KUKA KRL program: EPS_2_25694_LG02_A_20260223033039.src

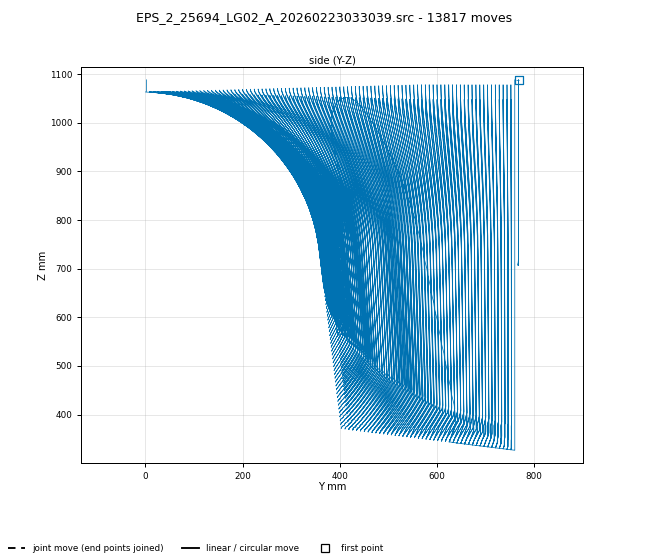
[picture p0: tool path of EPS_2_25694_LG02_A_20260223033039.src, 13817 of 13819 moves have a stored position in this frame; points joined in program order, loops and branches not executed]
&ACCESS RVP
&REL 4
&COMMENT QRS 19112012
&PARAM EDITMASK = *
DEF PART()
EXT BAS (BAS_COMMAND :IN,REAL :IN )
INT I
BAS (#INITMOV,0 )

;KUKA QRS Post kuka4.cps  Date:22-06-2017 !

File_ID=3045

QRS_PRE_INIT()

;Init var - Until changes are made in qrs_pre_init
Outlet_Square_prg=0
Inlet_1_Square_prg=0
Inlet_2_Square_prg=0
Inlet_3_Square_prg=0
Inlet_4_Square_prg=0
Inlet_5_Square_prg=0

Outlet_1={X 0.000, Y 562.000, Z 735.500, B 0.000, E1 0.000 }
Inlet_1={X 0.000, Y 562.000, Z 705.500, B 0.000, E1 182.000 }
Outlet_1_type=686
Inlet_1_type=686
;QRS#1=Sidecore dimensions
;QRS#2=675-27" Concrete
;QRS#3=675-27" Concrete
;QRS#4=
;QRS#5=
;QRS#6=
;QRS#7=
;QRS#8=
;QRS#9=S306-38L
;QRS#10=S306-38L
;QRS#11=
;QRS#12=
;QRS#13=
;QRS#14=
;QRS#15=
;QRS#16=1524x152x1524 5'
;QRS#17=EPS Height
;QRS#18=1078,5
;QRS#19=*
;QRS#20= UPDATED VERSION 22-06-2017
;QRS#21=*
Outlet_Square=0550
Inlet_1_Square=0550
Inlet_2_Square=0
Inlet_3_Square=0
Inlet_4_Square=0
Inlet_5_Square=0
Mill_Square=1
Outlet_Square_Prg=265
Inlet_1_Square_prg=265

QRS_INIT()

$ADVANCE=5

; T1
PTP {E1 173.043,E2 173.043}
PTP {X 0,Y 767.707,A -85,B 0,C 180,E1 173.043,E2 173.043,E3 0,E4 0,E5 0,E6 0}
QRS_SPEED_INIT()
LIN {X 0,Y 767.707,Z 1088.5,A -85,B 0,C 180,E1 173.043,E2 173.043,E3 0,E4 0,E5 0,E6 0} C_VEL
LIN {X 0,Y 767.707,Z 709.31,A -85,B 0,C 180,E1 173.043,E2 173.043} C_VEL
LIN {X 0,Y 767.734,Z 707.31,A -85,B 0,C 180,E1 173.192,E2 173.192} C_VEL
LIN {X 0,Y 767.794,Z 707.31,A -85,B 0,C 180,E1 173.458,E2 173.458} C_VEL
LIN {X 0,Y 767.812,Z 707.31,A -85,B 0,C 180,E1 177.201,E2 177.201} C_VEL
LIN {X 0,Y 767.838,Z 707.31,A -85,B 0,C 180,E1 180.933,E2 180.933} C_VEL
LIN {X 0,Y 767.834,Z 707.31,A -85,B 0,C 180,E1 184.668,E2 184.668} C_VEL
LIN {X 0,Y 767.857,Z 707.31,A -85,B 0,C 180,E1 188.423,E2 188.423} C_VEL
LIN {X 0,Y 767.828,Z 707.31,A -85,B 0,C 180,E1 192.215,E2 192.215} C_VEL
LIN {X 0,Y 767.83,Z 707.31,A -85,B 0,C 180,E1 196.204,E2 196.204} C_VEL
LIN {X 0,Y 767.77,Z 707.31,A -85,B 0,C 180,E1 199.988,E2 199.988} C_VEL
LIN {X 0,Y 767.749,Z 707.31,A -85,B 0,C 180,E1 204.013,E2 204.013} C_VEL
LIN {X 0,Y 767.749,Z 707.31,A -85,B 0,C 180,E1 208.167,E2 208.167} C_VEL
LIN {X 0,Y 767.324,Z 707.31,A -85,B 0,C 180,E1 210.324,E2 210.324} C_VEL
LIN {X 0,Y 767.754,Z 707.31,A -85,B 0,C 180,E1 212.49,E2 212.49} C_VEL
LIN {X 0,Y 767.43,Z 707.31,A -85,B 0,C 180,E1 213.85,E2 213.85} C_VEL
LIN {X 0,Y 767.706,Z 707.31,A -85,B 0,C 180,E1 217.094,E2 217.094} C_VEL
LIN {X 0,Y 767.087,Z 707.31,A -85,B 0,C 180,E1 220.03,E2 220.03} C_VEL
LIN {X 0,Y 767.533,Z 707.31,A -85,B 0,C 180,E1 221.88,E2 221.88} C_VEL
LIN {X 0,Y 767.581,Z 707.31,A -85,B 0,C 180,E1 222.891,E2 222.891} C_VEL
LIN {X 0,Y 767.581,Z 707.31,A -85,B 0,C 180,E1 227.109,E2 227.109} C_VEL
LIN {X 0,Y 767.53,Z 707.31,A -85,B 0,C 180,E1 228.12,E2 228.12} C_VEL
LIN {X 0,Y 767.102,Z 707.31,A -85,B 0,C 180,E1 230.553,E2 230.553} C_VEL
LIN {X 0,Y 767.692,Z 707.31,A -85,B 0,C 180,E1 232.964,E2 232.964} C_VEL
LIN {X 0,Y 767.598,Z 707.31,A -85,B 0,C 180,E1 236.132,E2 236.132} C_VEL
LIN {X 0,Y 767.614,Z 707.31,A -85,B 0,C 180,E1 237.503,E2 237.503} C_VEL
LIN {X 0,Y 767.641,Z 707.31,A -85,B 0,C 180,E1 239.69,E2 239.69} C_VEL
LIN {X 0,Y 767.411,Z 728.972,A -85,B 0,C 180,E1 240.873,E2 240.873} C_VEL
LIN {X 0,Y 767.537,Z 761.794,A -85,B 0,C 180,E1 241.233,E2 241.233} C_VEL
LIN {X 0,Y 767.433,Z 775.287,A -85,B 0,C 180,E1 241.407,E2 241.407} C_VEL
LIN {X 0,Y 767.548,Z 791.125,A -85,B 0,C 180,E1 241.677,E2 241.677} C_VEL
LIN {X 0,Y 767.449,Z 807.751,A -85,B 0,C 180,E1 242.019,E2 242.019} C_VEL
LIN {X 0,Y 767.663,Z 824.865,A -85,B 0,C 180,E1 242.456,E2 242.456} C_VEL
LIN {X 0,Y 767.66,Z 840.824,A -85,B 0,C 180,E1 242.921,E2 242.921} C_VEL
LIN {X 0,Y 767.553,Z 854.893,A -85,B 0,C 180,E1 243.38,E2 243.38} C_VEL
LIN {X 0,Y 767.694,Z 871.263,A -85,B 0,C 180,E1 243.998,E2 243.998} C_VEL
LIN {X 0,Y 767.655,Z 888.029,A -85,B 0,C 180,E1 244.706,E2 244.706} C_VEL
LIN {X 0,Y 767.705,Z 901.803,A -85,B 0,C 180,E1 245.351,E2 245.351} C_VEL
LIN {X 0,Y 767.712,Z 916.578,A -85,B 0,C 180,E1 246.114,E2 246.114} C_VEL
LIN {X 0,Y 767.693,Z 930.073,A -85,B 0,C 180,E1 246.876,E2 246.876} C_VEL
LIN {X 0,Y 767.691,Z 942.43,A -85,B 0,C 180,E1 247.634,E2 247.634} C_VEL
LIN {X 0,Y 767.701,Z 955.671,A -85,B 0,C 180,E1 248.523,E2 248.523} C_VEL
LIN {X 0,Y 767.718,Z 968.193,A -85,B 0,C 180,E1 249.439,E2 249.439} C_VEL
LIN {X 0,Y 767.619,Z 980.058,A -85,B 0,C 180,E1 250.38,E2 250.38} C_VEL
LIN {X 0,Y 767.656,Z 990.133,A -85,B 0,C 180,E1 251.245,E2 251.245} C_VEL
LIN {X 0,Y 767.778,Z 1000.684,A -85,B 0,C 180,E1 252.23,E2 252.23} C_VEL
LIN {X 0,Y 767.637,Z 1011.458,A -85,B 0,C 180,E1 253.326,E2 253.326} C_VEL
LIN {X 0,Y 767.699,Z 1020.421,A -85,B 0,C 180,E1 254.322,E2 254.322} C_VEL
LIN {X 0,Y 767.767,Z 1028.418,A -85,B 0,C 180,E1 255.29,E2 255.29} C_VEL
LIN {X 0,Y 767.624,Z 1037.824,A -85,B 0,C 180,E1 256.546,E2 256.546} C_VEL
LIN {X 0,Y 767.75,Z 1044.548,A -85,B 0,C 180,E1 257.545,E2 257.545} C_VEL
LIN {X 0,Y 767.749,Z 1048.907,A -85,B 0,C 180,E1 258.26,E2 258.26} C_VEL
LIN {X 0,Y 767.595,Z 1053.115,A -85,B 0,C 180,E1 258.971,E2 258.971} C_VEL
LIN {X 0,Y 767.579,Z 1059.347,A -85,B 0,C 180,E1 260.157,E2 260.157} C_VEL
LIN {X 0,Y 767.814,Z 1064.751,A -85,B 0,C 180,E1 261.341,E2 261.341} C_VEL
LIN {X 0,Y 767.552,Z 1069.482,A -85,B 0,C 180,E1 262.516,E2 262.516} C_VEL
LIN {X 0,Y 767.638,Z 1073.816,A -85,B 0,C 180,E1 263.832,E2 263.832} C_VEL
LIN {X 0,Y 767.832,Z 1075.822,A -85,B 0,C 180,E1 264.583,E2 264.583} C_VEL
LIN {X 0,Y 767.656,Z 1077.679,A -85,B 0,C 180,E1 265.331,E2 265.331} C_VEL
LIN {X 0,Y 767.554,Z 1079.934,A -85,B 0,C 180,E1 266.453,E2 266.453} C_VEL
LIN {X 0,Y 767.665,Z 1081.027,A -85,B 0,C 180,E1 267.201,E2 267.201} C_VEL
LIN {X 0,Y 767.713,Z 1082.196,A -85,B 0,C 180,E1 268.321,E2 268.321} C_VEL
LIN {X 0,Y 767.556,Z 1082.708,A -85,B 0,C 180,E1 269.067,E2 269.067} C_VEL
LIN {X 0,Y 767.7,Z 1082.68,A -85,B 0,C 180,E1 270.933,E2 270.933} C_VEL
LIN {X 0,Y 767.756,Z 1082.187,A -85,B 0,C 180,E1 271.679,E2 271.679} C_VEL
LIN {X 0,Y 767.525,Z 1081.053,A -85,B 0,C 180,E1 272.8,E2 272.8} C_VEL
LIN {X 0,Y 767.569,Z 1079.273,A -85,B 0,C 180,E1 273.921,E2 273.921} C_VEL
LIN {X 0,Y 767.76,Z 1077.66,A -85,B 0,C 180,E1 274.668,E2 274.668} C_VEL
LIN {X 0,Y 767.653,Z 1074.831,A -85,B 0,C 180,E1 275.793,E2 275.793} C_VEL
LIN {X 0,Y 767.602,Z 1072.628,A -85,B 0,C 180,E1 276.544,E2 276.544} C_VEL
LIN {X 0,Y 767.713,Z 1069.455,A -85,B 0,C 180,E1 277.483,E2 277.483} C_VEL
LIN {X 0,Y 767.824,Z 1067.577,A -85,B 0,C 180,E1 277.952,E2 277.952} C_VEL
LIN {X 0,Y 767.62,Z 1063.756,A -85,B 0,C 180,E1 278.897,E2 278.897} C_VEL
LIN {X 0,Y 767.559,Z 1058.195,A -85,B 0,C 180,E1 280.08,E2 280.08} C_VEL
LIN {X 0,Y 767.835,Z 1051.779,A -85,B 0,C 180,E1 281.263,E2 281.263} C_VEL
LIN {X 0,Y 767.624,Z 1044.562,A -85,B 0,C 180,E1 282.457,E2 282.457} C_VEL
LIN {X 0,Y 767.658,Z 1036.703,A -85,B 0,C 180,E1 283.612,E2 283.612} C_VEL
LIN {X 0,Y 767.821,Z 1029.879,A -85,B 0,C 180,E1 284.516,E2 284.516} C_VEL
LIN {X 0,Y 767.629,Z 1020.425,A -85,B 0,C 180,E1 285.679,E2 285.679} C_VEL
LIN {X 0,Y 767.731,Z 1009.175,A -85,B 0,C 180,E1 286.916,E2 286.916} C_VEL
LIN {X 0,Y 767.752,Z 999.435,A -85,B 0,C 180,E1 287.893,E2 287.893} C_VEL
LIN {X 0,Y 767.658,Z 988.765,A -85,B 0,C 180,E1 288.878,E2 288.878} C_VEL
LIN {X 0,Y 767.742,Z 977.061,A -85,B 0,C 180,E1 289.864,E2 289.864} C_VEL
LIN {X 0,Y 767.717,Z 964.937,A -85,B 0,C 180,E1 290.806,E2 290.806} C_VEL
LIN {X 0,Y 767.695,Z 954,A -85,B 0,C 180,E1 291.594,E2 291.594} C_VEL
LIN {X 0,Y 767.712,Z 940.407,A -85,B 0,C 180,E1 292.491,E2 292.491} C_VEL
LIN {X 0,Y 767.708,Z 926.801,A -85,B 0,C 180,E1 293.314,E2 293.314} C_VEL
LIN {X 0,Y 767.702,Z 913.125,A -85,B 0,C 180,E1 294.071,E2 294.071} C_VEL
LIN {X 0,Y 767.609,Z 898.313,A -85,B 0,C 180,E1 294.82,E2 294.82} C_VEL
LIN {X 0,Y 767.699,Z 884.655,A -85,B 0,C 180,E1 295.444,E2 295.444} C_VEL
LIN {X 0,Y 767.675,Z 869.452,A -85,B 0,C 180,E1 296.074,E2 296.074} C_VEL
LIN {X 0,Y 767.622,Z 855.716,A -85,B 0,C 180,E1 296.587,E2 296.587} C_VEL
LIN {X 0,Y 767.679,Z 837.478,A -85,B 0,C 180,E1 297.183,E2 297.183} C_VEL
LIN {X 0,Y 767.517,Z 820.546,A -85,B 0,C 180,E1 297.665,E2 297.665} C_VEL
LIN {X 0,Y 767.57,Z 810.446,A -85,B 0,C 180,E1 297.91,E2 297.91} C_VEL
LIN {X 0,Y 767.621,Z 801.596,A -85,B 0,C 180,E1 298.106,E2 298.106} C_VEL
LIN {X 0,Y 767.599,Z 787.938,A -85,B 0,C 180,E1 298.38,E2 298.38} C_VEL
LIN {X 0,Y 767.429,Z 775.319,A -85,B 0,C 180,E1 298.593,E2 298.593} C_VEL
LIN {X 0,Y 767.549,Z 757.089,A -85,B 0,C 180,E1 298.825,E2 298.825} C_VEL
LIN {X 0,Y 767.411,Z 729.388,A -85,B 0,C 180,E1 299.122,E2 299.122} C_VEL
LIN {X 0,Y 767.69,Z 707.31,A -85,B 0,C 180,E1 300.308,E2 300.308} C_VEL
LIN {X 0,Y 767.796,Z 707.31,A -85,B 0,C 180,E1 302.488,E2 302.488} C_VEL
LIN {X 0,Y 767.259,Z 707.31,A -85,B 0,C 180,E1 304.756,E2 304.756} C_VEL
LIN {X 0,Y 767.698,Z 707.31,A -85,B 0,C 180,E1 307.093,E2 307.093} C_VEL
LIN {X 0,Y 767.134,Z 707.31,A -85,B 0,C 180,E1 310.034,E2 310.034} C_VEL
LIN {X 0,Y 767.63,Z 707.31,A -85,B 0,C 180,E1 311.873,E2 311.873} C_VEL
LIN {X 0,Y 767.669,Z 707.31,A -85,B 0,C 180,E1 312.898,E2 312.898} C_VEL
LIN {X 0,Y 767.67,Z 707.31,A -85,B 0,C 180,E1 314.427,E2 314.427} C_VEL
LIN {X 0,Y 767.632,Z 707.31,A -85,B 0,C 180,E1 315.57,E2 315.57} C_VEL
LIN {X 0,Y 767.641,Z 707.31,A -85,B 0,C 180,E1 319.92,E2 319.92} C_VEL
LIN {X 0,Y 767.641,Z 707.31,A -85,B 0,C 180,E1 320.586,E2 320.586} C_VEL
LIN {X 0,Y 767.2,Z 707.31,A -85,B 0,C 180,E1 322.956,E2 322.956} C_VEL
LIN {X 0,Y 767.714,Z 707.31,A -85,B 0,C 180,E1 325.268,E2 325.268} C_VEL
LIN {X 0,Y 767.762,Z 707.31,A -85,B 0,C 180,E1 329.62,E2 329.62} C_VEL
LIN {X 0,Y 767.769,Z 707.31,A -85,B 0,C 180,E1 333.539,E2 333.539} C_VEL
LIN {X 0,Y 767.759,Z 707.31,A -85,B 0,C 180,E1 333.929,E2 333.929} C_VEL
LIN {X 0,Y 767.758,Z 707.31,A -85,B 0,C 180,E1 338.014,E2 338.014} C_VEL
LIN {X 0,Y 767.79,Z 707.31,A -85,B 0,C 180,E1 341.986,E2 341.986} C_VEL
LIN {X 0,Y 767.525,Z 707.31,A -85,B 0,C 180,E1 343.931,E2 343.931} C_VEL
LIN {X 0,Y 767.673,Z 707.31,A -85,B 0,C 180,E1 345.866,E2 345.866} C_VEL
LIN {X 0,Y 767.85,Z 707.31,A -85,B 0,C 180,E1 349.687,E2 349.687} C_VEL
LIN {X 0,Y 767.871,Z 707.31,A -85,B 0,C 180,E1 353.458,E2 353.458} C_VEL
LIN {X 0,Y 767.845,Z 707.31,A -85,B 0,C 180,E1 357.201,E2 357.201} C_VEL
LIN {X 0,Y 767.813,Z 707.31,A -85,B 0,C 180,E1 360.933,E2 360.933} C_VEL
LIN {X 0,Y 767.808,Z 707.31,A -85,B 0,C 180,E1 364.668,E2 364.668} C_VEL
LIN {X 0,Y 767.797,Z 707.31,A -85,B 0,C 180,E1 368.424,E2 368.424} C_VEL
LIN {X 0,Y 767.811,Z 707.31,A -85,B 0,C 180,E1 372.216,E2 372.216} C_VEL
LIN {X 0,Y 767.847,Z 707.31,A -85,B 0,C 180,E1 376.209,E2 376.209} C_VEL
LIN {X 0,Y 767.467,Z 707.31,A -85,B 0,C 180,E1 379.996,E2 379.996} C_VEL
LIN {X 0,Y 767.321,Z 707.31,A -85,B 0,C 180,E1 381.999,E2 381.999} C_VEL
LIN {X 0,Y 767.24,Z 707.31,A -85,B 0,C 180,E1 384.03,E2 384.03} C_VEL
LIN {X 0,Y 767.58,Z 707.31,A -85,B 0,C 180,E1 386.078,E2 386.078} C_VEL
LIN {X 0,Y 767.754,Z 707.31,A -85,B 0,C 180,E1 390.379,E2 390.379} C_VEL
LIN {X 0,Y 767.374,Z 707.31,A -85,B 0,C 180,E1 393.844,E2 393.844} C_VEL
LIN {X 0,Y 767.676,Z 707.31,A -85,B 0,C 180,E1 394.734,E2 394.734} C_VEL
LIN {X 0,Y 767.196,Z 707.31,A -85,B 0,C 180,E1 397.064,E2 397.064} C_VEL
LIN {X 0,Y 767.661,Z 707.31,A -85,B 0,C 180,E1 399.412,E2 399.412} C_VEL
LIN {X 0,Y 767.663,Z 707.31,A -85,B 0,C 180,E1 400.082,E2 400.082} C_VEL
LIN {X 0,Y 767.636,Z 707.31,A -85,B 0,C 180,E1 404.43,E2 404.43} C_VEL
LIN {X 0,Y 767.465,Z 707.31,A -85,B 0,C 180,E1 405.558,E2 405.558} C_VEL
LIN {X 0,Y 767.675,Z 707.31,A -85,B 0,C 180,E1 409.918,E2 409.918} C_VEL
LIN {X 0,Y 767.742,Z 707.31,A -85,B 0,C 180,E1 410.593,E2 410.593} C_VEL
LIN {X 0,Y 767.651,Z 707.31,A -85,B 0,C 180,E1 412.962,E2 412.962} C_VEL
LIN {X 0,Y 767.133,Z 707.31,A -85,B 0,C 180,E1 415.238,E2 415.238} C_VEL
LIN {X 0,Y 767.859,Z 707.31,A -85,B 0,C 180,E1 418.652,E2 418.652} C_VEL
LIN {X 0,Y 766.583,Z 707.31,A -85,B 0,C 180,E1 418.851,E2 418.851} C_VEL
LIN {X 0,Y 766.332,Z 707.453,A -85,B 0,C 180,E1 418.872,E2 418.872} C_VEL
LIN {X 0,Y 767.228,Z 716.962,A -85,B 0,C 180,E1 419.009,E2 419.009} C_VEL
LIN {X 0,Y 767.514,Z 728.846,A -85,B 0,C 180,E1 419.15,E2 419.15} C_VEL
LIN {X 0,Y 767.577,Z 744.469,A -85,B 0,C 180,E1 419.354,E2 419.354} C_VEL
LIN {X 0,Y 767.448,Z 760.576,A -85,B 0,C 180,E1 419.617,E2 419.617} C_VEL
LIN {X 0,Y 767.544,Z 778.604,A -85,B 0,C 180,E1 419.999,E2 419.999} C_VEL
LIN {X 0,Y 767.515,Z 791.795,A -85,B 0,C 180,E1 420.32,E2 420.32} C_VEL
LIN {X 0,Y 767.646,Z 810.803,A -85,B 0,C 180,E1 420.875,E2 420.875} C_VEL
LIN {X 0,Y 767.539,Z 825.708,A -85,B 0,C 180,E1 421.364,E2 421.364} C_VEL
LIN {X 0,Y 767.659,Z 841.503,A -85,B 0,C 180,E1 421.961,E2 421.961} C_VEL
LIN {X 0,Y 767.652,Z 857.144,A -85,B 0,C 180,E1 422.619,E2 422.619} C_VEL
LIN {X 0,Y 767.699,Z 872.8,A -85,B 0,C 180,E1 423.357,E2 423.357} C_VEL
LIN {X 0,Y 767.696,Z 886.598,A -85,B 0,C 180,E1 424.069,E2 424.069} C_VEL
LIN {X 0,Y 767.675,Z 900.841,A -85,B 0,C 180,E1 424.877,E2 424.877} C_VEL
LIN {X 0,Y 767.698,Z 912.552,A -85,B 0,C 180,E1 425.598,E2 425.598} C_VEL
LIN {X 0,Y 767.712,Z 925.914,A -85,B 0,C 180,E1 426.496,E2 426.496} C_VEL
LIN {X 0,Y 767.737,Z 938.055,A -85,B 0,C 180,E1 427.383,E2 427.383} C_VEL
LIN {X 0,Y 767.685,Z 949.6,A -85,B 0,C 180,E1 428.298,E2 428.298} C_VEL
LIN {X 0,Y 767.77,Z 960.082,A -85,B 0,C 180,E1 429.198,E2 429.198} C_VEL
LIN {X 0,Y 767.697,Z 971.428,A -85,B 0,C 180,E1 430.258,E2 430.258} C_VEL
LIN {X 0,Y 767.651,Z 981.132,A -85,B 0,C 180,E1 431.245,E2 431.245} C_VEL
LIN {X 0,Y 767.822,Z 991.022,A -85,B 0,C 180,E1 432.354,E2 432.354} C_VEL
LIN {X 0,Y 767.594,Z 999.985,A -85,B 0,C 180,E1 433.446,E2 433.446} C_VEL
LIN {X 0,Y 767.611,Z 1007.914,A -85,B 0,C 180,E1 434.514,E2 434.514} C_VEL
LIN {X 0,Y 767.808,Z 1015.644,A -85,B 0,C 180,E1 435.676,E2 435.676} C_VEL
LIN {X 0,Y 767.569,Z 1022.576,A -85,B 0,C 180,E1 436.824,E2 436.824} C_VEL
LIN {X 0,Y 767.623,Z 1028.911,A -85,B 0,C 180,E1 438.02,E2 438.02} C_VEL
LIN {X 0,Y 767.827,Z 1033.324,A -85,B 0,C 180,E1 438.975,E2 438.975} C_VEL
LIN {X 0,Y 767.639,Z 1036.336,A -85,B 0,C 180,E1 439.684,E2 439.684} C_VEL
LIN {X 0,Y 767.554,Z 1040.012,A -85,B 0,C 180,E1 440.63,E2 440.63} C_VEL
LIN {X 0,Y 767.677,Z 1043.168,A -85,B 0,C 180,E1 441.575,E2 441.575} C_VEL
LIN {X 0,Y 767.804,Z 1044.49,A -85,B 0,C 180,E1 442.048,E2 442.048} C_VEL
LIN {X 0,Y 767.778,Z 1045.777,A -85,B 0,C 180,E1 442.518,E2 442.518} C_VEL
LIN {X 0,Y 767.584,Z 1048.049,A -85,B 0,C 180,E1 443.456,E2 443.456} C_VEL
LIN {X 0,Y 767.578,Z 1049.627,A -85,B 0,C 180,E1 444.207,E2 444.207} C_VEL
LIN {X 0,Y 767.792,Z 1051.269,A -85,B 0,C 180,E1 445.332,E2 445.332} C_VEL
LIN {X 0,Y 767.688,Z 1052.025,A -85,B 0,C 180,E1 446.08,E2 446.08} C_VEL
LIN {X 0,Y 767.517,Z 1052.766,A -85,B 0,C 180,E1 447.2,E2 447.2} C_VEL
LIN {X 0,Y 767.839,Z 1052.603,A -85,B 0,C 180,E1 449.067,E2 449.067} C_VEL
LIN {X 0,Y 767.684,Z 1051.712,A -85,B 0,C 180,E1 450.187,E2 450.187} C_VEL
LIN {X 0,Y 767.839,Z 1049.617,A -85,B 0,C 180,E1 451.679,E2 451.679} C_VEL
LIN {X 0,Y 767.587,Z 1047.326,A -85,B 0,C 180,E1 452.8,E2 452.8} C_VEL
LIN {X 0,Y 767.682,Z 1043.303,A -85,B 0,C 180,E1 454.295,E2 454.295} C_VEL
LIN {X 0,Y 767.813,Z 1040.757,A -85,B 0,C 180,E1 455.042,E2 455.042} C_VEL
LIN {X 0,Y 767.73,Z 1039.519,A -85,B 0,C 180,E1 455.417,E2 455.417} C_VEL
LIN {X 0,Y 767.568,Z 1034.048,A -85,B 0,C 180,E1 456.792,E2 456.792} C_VEL
LIN {X 0,Y 767.782,Z 1028.581,A -85,B 0,C 180,E1 457.953,E2 457.953} C_VEL
LIN {X 0,Y 767.744,Z 1024.81,A -85,B 0,C 180,E1 458.66,E2 458.66} C_VEL
LIN {X 0,Y 767.59,Z 1020.908,A -85,B 0,C 180,E1 459.37,E2 459.37} C_VEL
LIN {X 0,Y 767.566,Z 1015.193,A -85,B 0,C 180,E1 460.317,E2 460.317} C_VEL
LIN {X 0,Y 767.802,Z 1007.156,A -85,B 0,C 180,E1 461.501,E2 461.501} C_VEL
LIN {X 0,Y 767.587,Z 998.194,A -85,B 0,C 180,E1 462.697,E2 462.697} C_VEL
LIN {X 0,Y 767.586,Z 989.678,A -85,B 0,C 180,E1 463.725,E2 463.725} C_VEL
LIN {X 0,Y 767.795,Z 978.848,A -85,B 0,C 180,E1 464.902,E2 464.902} C_VEL
LIN {X 0,Y 767.649,Z 968.142,A -85,B 0,C 180,E1 465.97,E2 465.97} C_VEL
LIN {X 0,Y 767.685,Z 957.768,A -85,B 0,C 180,E1 466.917,E2 466.917} C_VEL
LIN {X 0,Y 767.774,Z 947.684,A -85,B 0,C 180,E1 467.77,E2 467.77} C_VEL
LIN {X 0,Y 767.697,Z 935.041,A -85,B 0,C 180,E1 468.754,E2 468.754} C_VEL
LIN {X 0,Y 767.717,Z 922.969,A -85,B 0,C 180,E1 469.617,E2 469.617} C_VEL
LIN {X 0,Y 767.739,Z 910.052,A -85,B 0,C 180,E1 470.467,E2 470.467} C_VEL
LIN {X 0,Y 767.713,Z 896.37,A -85,B 0,C 180,E1 471.293,E2 471.293} C_VEL
LIN {X 0,Y 767.691,Z 882.652,A -85,B 0,C 180,E1 472.051,E2 472.051} C_VEL
LIN {X 0,Y 767.715,Z 868.914,A -85,B 0,C 180,E1 472.744,E2 472.744} C_VEL
LIN {X 0,Y 767.701,Z 853.646,A -85,B 0,C 180,E1 473.441,E2 473.441} C_VEL
LIN {X 0,Y 767.559,Z 838.183,A -85,B 0,C 180,E1 474.081,E2 474.081} C_VEL
LIN {X 0,Y 767.686,Z 823.019,A -85,B 0,C 180,E1 474.632,E2 474.632} C_VEL
LIN {X 0,Y 767.65,Z 807.174,A -85,B 0,C 180,E1 475.148,E2 475.148} C_VEL
LIN {X 0,Y 767.562,Z 793.513,A -85,B 0,C 180,E1 475.542,E2 475.542} C_VEL
LIN {X 0,Y 767.685,Z 773.931,A -85,B 0,C 180,E1 476.011,E2 476.011} C_VEL
LIN {X 0,Y 767.51,Z 756.999,A -85,B 0,C 180,E1 476.354,E2 476.354} C_VEL
LIN {X 0,Y 767.504,Z 749.285,A -85,B 0,C 180,E1 476.48,E2 476.48} C_VEL
LIN {X 0,Y 767.595,Z 739.533,A -85,B 0,C 180,E1 476.623,E2 476.623} C_VEL
LIN {X 0,Y 767.474,Z 719.835,A -85,B 0,C 180,E1 476.861,E2 476.861} C_VEL
LIN {X 0,Y 767.332,Z 713.145,A -85,B 0,C 180,E1 476.936,E2 476.936} C_VEL
LIN {X 0,Y 766.479,Z 708.854,A -85,B 0,C 180,E1 477.017,E2 477.017} C_VEL
LIN {X 0,Y 766.257,Z 707.31,A -85,B 0,C 180,E1 477.063,E2 477.063} C_VEL
LIN {X 0,Y 766.793,Z 707.31,A -85,B 0,C 180,E1 477.102,E2 477.102} C_VEL
LIN {X 0,Y 767.511,Z 707.31,A -85,B 0,C 180,E1 477.191,E2 477.191} C_VEL
LIN {X 0,Y 767.758,Z 707.31,A -85,B 0,C 180,E1 477.693,E2 477.693} C_VEL
LIN {X 0,Y 767.795,Z 707.31,A -85,B 0,C 180,E1 480.384,E2 480.384} C_VEL
LIN {X 0,Y 767.697,Z 707.31,A -85,B 0,C 180,E1 484.733,E2 484.733} C_VEL
LIN {X 0,Y 767.22,Z 707.31,A -85,B 0,C 180,E1 487.062,E2 487.062} C_VEL
LIN {X 0,Y 767.7,Z 707.31,A -85,B 0,C 180,E1 489.41,E2 489.41} C_VEL
LIN {X 0,Y 767.687,Z 707.31,A -85,B 0,C 180,E1 490.084,E2 490.084} C_VEL
LIN {X 0,Y 767.469,Z 707.31,A -85,B 0,C 180,E1 494.442,E2 494.442} C_VEL
LIN {X 0,Y 767.64,Z 707.31,A -85,B 0,C 180,E1 495.57,E2 495.57} C_VEL
LIN {X 0,Y 767.663,Z 707.31,A -85,B 0,C 180,E1 499.919,E2 499.919} C_VEL
LIN {X 0,Y 767.648,Z 707.31,A -85,B 0,C 180,E1 500.587,E2 500.587} C_VEL
LIN {X 0,Y 767.199,Z 707.31,A -85,B 0,C 180,E1 502.956,E2 502.956} C_VEL
LIN {X 0,Y 767.684,Z 707.31,A -85,B 0,C 180,E1 505.266,E2 505.266} C_VEL
LIN {X 0,Y 767.764,Z 707.31,A -85,B 0,C 180,E1 509.62,E2 509.62} C_VEL
LIN {X 0,Y 767.79,Z 707.31,A -85,B 0,C 180,E1 513.536,E2 513.536} C_VEL
LIN {X 0,Y 767.787,Z 707.31,A -85,B 0,C 180,E1 513.93,E2 513.93} C_VEL
LIN {X 0,Y 767.808,Z 707.31,A -85,B 0,C 180,E1 518.016,E2 518.016} C_VEL
LIN {X 0,Y 767.827,Z 707.31,A -85,B 0,C 180,E1 521.986,E2 521.986} C_VEL
LIN {X 0,Y 767.5,Z 707.31,A -85,B 0,C 180,E1 523.93,E2 523.93} C_VEL
LIN {X 0,Y 767.615,Z 707.31,A -85,B 0,C 180,E1 525.865,E2 525.865} C_VEL
LIN {X 0,Y 767.793,Z 707.31,A -85,B 0,C 180,E1 529.686,E2 529.686} C_VEL
LIN {X 0,Y 767.734,Z 707.31,A -85,B 0,C 180,E1 533.192,E2 533.192} C_VEL
LIN {X 0,Y 767.795,Z 709.31,A -85,B 0,C 180,E1 533.341,E2 533.341} C_VEL
LIN {X 0,Y 767.795,Z 1088.5,A -85,B 0,C 180,E1 533.341,E2 533.341} C_VEL
LIN {X 0,Y 767.795,Z 1088.5,A -85,B 0,C 180,E1 533.341,E2 533.341}

QRS_NEXT_CUT()
PTP {E1 537.319,E2 537.319}
PTP {X 0,Y 759.843,A -85,B 0,C 180,E1 537.319,E2 537.319,E3 0,E4 0,E5 0,E6 0}
QRS_SPEED_INIT()
LIN {X 0,Y 759.843,Z 1088.5,A -85,B 0,C 180,E1 537.319,E2 537.319,E3 0,E4 0,E5 0,E6 0} C_VEL
LIN {X 0,Y 759.843,Z 336.65,A -85,B 0,C 180,E1 537.319,E2 537.319} C_VEL
LIN {X 0,Y 759.843,Z 328.572,A -85,B 0,C 180,E1 537.319,E2 537.319} C_VEL
LIN {X 0,Y 759.843,Z 326.572,A -85,B 0,C 180,E1 537.169,E2 537.169} C_VEL
LIN {X 0,Y 759.893,Z 326.569,A -85,B 0,C 180,E1 534.564,E2 534.564} C_VEL
LIN {X 0,Y 759.866,Z 326.575,A -85,B 0,C 180,E1 531.601,E2 531.601} C_VEL
LIN {X 0,Y 759.843,Z 326.572,A -85,B 0,C 180,E1 529.077,E2 529.077} C_VEL
LIN {X 0,Y 759.889,Z 326.569,A -85,B 0,C 180,E1 526.454,E2 526.454} C_VEL
LIN {X 0,Y 759.869,Z 326.575,A -85,B 0,C 180,E1 523.487,E2 523.487} C_VEL
LIN {X 0,Y 759.844,Z 326.572,A -85,B 0,C 180,E1 520.953,E2 520.953} C_VEL
LIN {X 0,Y 759.881,Z 326.569,A -85,B 0,C 180,E1 518.381,E2 518.381} C_VEL
LIN {X 0,Y 759.869,Z 326.575,A -85,B 0,C 180,E1 515.346,E2 515.346} C_VEL
LIN {X 0,Y 759.844,Z 326.572,A -85,B 0,C 180,E1 512.818,E2 512.818} C_VEL
LIN {X 0,Y 759.879,Z 326.569,A -85,B 0,C 180,E1 510.259,E2 510.259} C_VEL
LIN {X 0,Y 759.872,Z 326.575,A -85,B 0,C 180,E1 507.229,E2 507.229} C_VEL
LIN {X 0,Y 759.845,Z 326.572,A -85,B 0,C 180,E1 504.673,E2 504.673} C_VEL
LIN {X 0,Y 759.898,Z 326.568,A -85,B 0,C 180,E1 501.989,E2 501.989} C_VEL
LIN {X 0,Y 759.869,Z 326.575,A -85,B 0,C 180,E1 499.052,E2 499.052} C_VEL
LIN {X 0,Y 759.846,Z 326.571,A -85,B 0,C 180,E1 496.51,E2 496.51} C_VEL
LIN {X 0,Y 759.898,Z 326.568,A -85,B 0,C 180,E1 493.857,E2 493.857} C_VEL
LIN {X 0,Y 759.873,Z 326.576,A -85,B 0,C 180,E1 490.942,E2 490.942} C_VEL
LIN {X 0,Y 759.846,Z 326.573,A -85,B 0,C 180,E1 488.397,E2 488.397} C_VEL
LIN {X 0,Y 759.894,Z 326.569,A -85,B 0,C 180,E1 485.748,E2 485.748} C_VEL
LIN {X 0,Y 759.868,Z 326.579,A -85,B 0,C 180,E1 482.77,E2 482.77} C_VEL
LIN {X 0,Y 759.846,Z 326.656,A -85,B 0,C 180,E1 482.25,E2 482.25} C_VEL
LIN {X 0,Y 759.884,Z 347.643,A -85,B 0,C 180,E1 480.755,E2 480.755} C_VEL
LIN {X 0,Y 759.912,Z 584.911,A -85,B 0,C 180,E1 478.177,E2 478.177} C_VEL
LIN {X 0,Y 759.916,Z 736.017,A -85,B 0,C 180,E1 476.55,E2 476.55} C_VEL
LIN {X 0,Y 759.9,Z 759.461,A -85,B 0,C 180,E1 476.182,E2 476.182} C_VEL
LIN {X 0,Y 759.903,Z 781.523,A -85,B 0,C 180,E1 475.701,E2 475.701} C_VEL
LIN {X 0,Y 759.898,Z 801.218,A -85,B 0,C 180,E1 475.172,E2 475.172} C_VEL
LIN {X 0,Y 759.919,Z 824.386,A -85,B 0,C 180,E1 474.421,E2 474.421} C_VEL
LIN {X 0,Y 759.916,Z 844.946,A -85,B 0,C 180,E1 473.619,E2 473.619} C_VEL
LIN {X 0,Y 759.913,Z 864.955,A -85,B 0,C 180,E1 472.724,E2 472.724} C_VEL
LIN {X 0,Y 759.91,Z 887,A -85,B 0,C 180,E1 471.578,E2 471.578} C_VEL
LIN {X 0,Y 759.916,Z 905.657,A -85,B 0,C 180,E1 470.471,E2 470.471} C_VEL
LIN {X 0,Y 759.908,Z 925.564,A -85,B 0,C 180,E1 469.125,E2 469.125} C_VEL
LIN {X 0,Y 759.913,Z 942.712,A -85,B 0,C 180,E1 467.814,E2 467.814} C_VEL
LIN {X 0,Y 759.912,Z 959.488,A -85,B 0,C 180,E1 466.355,E2 466.355} C_VEL
LIN {X 0,Y 759.897,Z 973.888,A -85,B 0,C 180,E1 464.946,E2 464.946} C_VEL
LIN {X 0,Y 759.908,Z 988.501,A -85,B 0,C 180,E1 463.313,E2 463.313} C_VEL
LIN {X 0,Y 759.906,Z 1000.009,A -85,B 0,C 180,E1 461.845,E2 461.845} C_VEL
LIN {X 0,Y 759.912,Z 1012.038,A -85,B 0,C 180,E1 460.079,E2 460.079} C_VEL
LIN {X 0,Y 759.9,Z 1021.248,A -85,B 0,C 180,E1 458.475,E2 458.475} C_VEL
LIN {X 0,Y 759.894,Z 1029.42,A -85,B 0,C 180,E1 456.801,E2 456.801} C_VEL
LIN {X 0,Y 759.914,Z 1036.478,A -85,B 0,C 180,E1 454.982,E2 454.982} C_VEL
LIN {X 0,Y 759.893,Z 1041.296,A -85,B 0,C 180,E1 453.395,E2 453.395} C_VEL
LIN {X 0,Y 759.914,Z 1045.436,A -85,B 0,C 180,E1 451.508,E2 451.508} C_VEL
LIN {X 0,Y 759.902,Z 1047.622,A -85,B 0,C 180,E1 449.774,E2 449.774} C_VEL
LIN {X 0,Y 759.911,Z 1048.5,A -85,B 0,C 180,E1 447.964,E2 447.964} C_VEL
LIN {X 0,Y 759.903,Z 1047.636,A -85,B 0,C 180,E1 446.152,E2 446.152} C_VEL
LIN {X 0,Y 759.912,Z 1045.563,A -85,B 0,C 180,E1 444.488,E2 444.488} C_VEL
LIN {X 0,Y 759.895,Z 1041.501,A -85,B 0,C 180,E1 442.591,E2 442.591} C_VEL
LIN {X 0,Y 759.914,Z 1036.69,A -85,B 0,C 180,E1 440.992,E2 440.992} C_VEL
LIN {X 0,Y 759.893,Z 1029.632,A -85,B 0,C 180,E1 439.154,E2 439.154} C_VEL
LIN {X 0,Y 759.904,Z 1021.383,A -85,B 0,C 180,E1 437.461,E2 437.461} C_VEL
LIN {X 0,Y 759.912,Z 1012.276,A -85,B 0,C 180,E1 435.871,E2 435.871} C_VEL
LIN {X 0,Y 759.907,Z 1000.391,A -85,B 0,C 180,E1 434.116,E2 434.116} C_VEL
LIN {X 0,Y 759.908,Z 988.697,A -85,B 0,C 180,E1 432.621,E2 432.621} C_VEL
LIN {X 0,Y 759.903,Z 973.001,A -85,B 0,C 180,E1 430.875,E2 430.875} C_VEL
LIN {X 0,Y 759.909,Z 959.029,A -85,B 0,C 180,E1 429.512,E2 429.512} C_VEL
LIN {X 0,Y 759.915,Z 940.673,A -85,B 0,C 180,E1 427.935,E2 427.935} C_VEL
LIN {X 0,Y 759.917,Z 923.41,A -85,B 0,C 180,E1 426.627,E2 426.627} C_VEL
LIN {X 0,Y 759.914,Z 903.513,A -85,B 0,C 180,E1 425.306,E2 425.306} C_VEL
LIN {X 0,Y 759.91,Z 885.071,A -85,B 0,C 180,E1 424.223,E2 424.223} C_VEL
LIN {X 0,Y 759.915,Z 862.835,A -85,B 0,C 180,E1 423.087,E2 423.087} C_VEL
LIN {X 0,Y 759.918,Z 843.709,A -85,B 0,C 180,E1 422.239,E2 422.239} C_VEL
LIN {X 0,Y 759.913,Z 820.69,A -85,B 0,C 180,E1 421.359,E2 421.359} C_VEL
LIN {X 0,Y 759.903,Z 799.673,A -85,B 0,C 180,E1 420.693,E2 420.693} C_VEL
LIN {X 0,Y 759.9,Z 779.134,A -85,B 0,C 180,E1 420.15,E2 420.15} C_VEL
LIN {X 0,Y 759.908,Z 753.73,A -85,B 0,C 180,E1 419.629,E2 419.629} C_VEL
LIN {X 0,Y 759.917,Z 733.55,A -85,B 0,C 180,E1 419.329,E2 419.329} C_VEL
LIN {X 0,Y 759.917,Z 462.351,A -85,B 0,C 180,E1 416.411,E2 416.411} C_VEL
LIN {X 0,Y 759.883,Z 347.478,A -85,B 0,C 180,E1 415.152,E2 415.152} C_VEL
LIN {X 0,Y 759.844,Z 326.576,A -85,B 0,C 180,E1 413.644,E2 413.644} C_VEL
LIN {X 0,Y 759.867,Z 326.576,A -85,B 0,C 180,E1 411.121,E2 411.121} C_VEL
LIN {X 0,Y 759.892,Z 326.569,A -85,B 0,C 180,E1 408.139,E2 408.139} C_VEL
LIN {X 0,Y 759.844,Z 326.572,A -85,B 0,C 180,E1 405.498,E2 405.498} C_VEL
LIN {X 0,Y 759.868,Z 326.575,A -85,B 0,C 180,E1 402.971,E2 402.971} C_VEL
LIN {X 0,Y 759.884,Z 326.569,A -85,B 0,C 180,E1 399.951,E2 399.951} C_VEL
LIN {X 0,Y 759.843,Z 326.573,A -85,B 0,C 180,E1 397.347,E2 397.347} C_VEL
LIN {X 0,Y 759.87,Z 326.574,A -85,B 0,C 180,E1 394.805,E2 394.805} C_VEL
LIN {X 0,Y 759.877,Z 326.569,A -85,B 0,C 180,E1 391.759,E2 391.759} C_VEL
LIN {X 0,Y 759.843,Z 326.572,A -85,B 0,C 180,E1 389.223,E2 389.223} C_VEL
LIN {X 0,Y 759.868,Z 326.575,A -85,B 0,C 180,E1 386.686,E2 386.686} C_VEL
LIN {X 0,Y 759.882,Z 326.569,A -85,B 0,C 180,E1 383.662,E2 383.662} C_VEL
LIN {X 0,Y 759.842,Z 326.572,A -85,B 0,C 180,E1 381.054,E2 381.054} C_VEL
LIN {X 0,Y 759.865,Z 326.575,A -85,B 0,C 180,E1 378.569,E2 378.569} C_VEL
LIN {X 0,Y 759.888,Z 326.569,A -85,B 0,C 180,E1 375.571,E2 375.571} C_VEL
LIN {X 0,Y 759.843,Z 326.572,A -85,B 0,C 180,E1 373.004,E2 373.004} C_VEL
LIN {X 0,Y 759.855,Z 326.575,A -85,B 0,C 180,E1 370.539,E2 370.539} C_VEL
LIN {X 0,Y 759.916,Z 326.569,A -85,B 0,C 180,E1 367.637,E2 367.637} C_VEL
LIN {X 0,Y 759.844,Z 326.572,A -85,B 0,C 180,E1 364.907,E2 364.907} C_VEL
LIN {X 0,Y 759.854,Z 326.575,A -85,B 0,C 180,E1 362.413,E2 362.413} C_VEL
LIN {X 0,Y 759.918,Z 326.57,A -85,B 0,C 180,E1 359.548,E2 359.548} C_VEL
LIN {X 0,Y 759.846,Z 326.571,A -85,B 0,C 180,E1 356.832,E2 356.832} C_VEL
LIN {X 0,Y 759.849,Z 326.574,A -85,B 0,C 180,E1 354.336,E2 354.336} C_VEL
LIN {X 0,Y 759.916,Z 326.572,A -85,B 0,C 180,E1 351.525,E2 351.525} C_VEL
LIN {X 0,Y 759.849,Z 326.571,A -85,B 0,C 180,E1 348.77,E2 348.77} C_VEL
LIN {X 0,Y 759.844,Z 326.574,A -85,B 0,C 180,E1 346.298,E2 346.298} C_VEL
LIN {X 0,Y 759.915,Z 326.577,A -85,B 0,C 180,E1 343.567,E2 343.567} C_VEL
LIN {X 0,Y 759.853,Z 326.571,A -85,B 0,C 180,E1 340.713,E2 340.713} C_VEL
LIN {X 0,Y 759.84,Z 326.573,A -85,B 0,C 180,E1 338.286,E2 338.286} C_VEL
LIN {X 0,Y 759.872,Z 326.575,A -85,B 0,C 180,E1 335.76,E2 335.76} C_VEL
LIN {X 0,Y 759.872,Z 326.57,A -85,B 0,C 180,E1 332.747,E2 332.747} C_VEL
LIN {X 0,Y 759.84,Z 326.573,A -85,B 0,C 180,E1 330.257,E2 330.257} C_VEL
LIN {X 0,Y 759.854,Z 326.575,A -85,B 0,C 180,E1 327.792,E2 327.792} C_VEL
LIN {X 0,Y 759.91,Z 326.57,A -85,B 0,C 180,E1 324.9,E2 324.9} C_VEL
LIN {X 0,Y 759.845,Z 326.572,A -85,B 0,C 180,E1 322.266,E2 322.266} C_VEL
LIN {X 0,Y 759.842,Z 326.574,A -85,B 0,C 180,E1 319.849,E2 319.849} C_VEL
LIN {X 0,Y 759.909,Z 326.578,A -85,B 0,C 180,E1 317.13,E2 317.13} C_VEL
LIN {X 0,Y 759.855,Z 326.571,A -85,B 0,C 180,E1 314.287,E2 314.287} C_VEL
LIN {X 0,Y 759.839,Z 326.574,A -85,B 0,C 180,E1 311.849,E2 311.849} C_VEL
LIN {X 0,Y 759.877,Z 326.577,A -85,B 0,C 180,E1 309.266,E2 309.266} C_VEL
LIN {X 0,Y 759.863,Z 326.573,A -85,B 0,C 180,E1 306.231,E2 306.231} C_VEL
LIN {X 0,Y 759.857,Z 326.883,A -85,B 0,C 180,E1 306.17,E2 306.17} C_VEL
LIN {X 0,Y 759.903,Z 363.722,A -85,B 0,C 180,E1 303.684,E2 303.684} C_VEL
LIN {X 0,Y 759.914,Z 377.344,A -85,B 0,C 180,E1 302.802,E2 302.802} C_VEL
LIN {X 0,Y 759.918,Z 632.42,A -85,B 0,C 180,E1 300.034,E2 300.034} C_VEL
LIN {X 0,Y 759.915,Z 765.994,A -85,B 0,C 180,E1 298.595,E2 298.595} C_VEL
LIN {X 0,Y 759.897,Z 790.301,A -85,B 0,C 180,E1 298.21,E2 298.21} C_VEL
LIN {X 0,Y 759.902,Z 811.683,A -85,B 0,C 180,E1 297.742,E2 297.742} C_VEL
LIN {X 0,Y 759.901,Z 831.086,A -85,B 0,C 180,E1 297.221,E2 297.221} C_VEL
LIN {X 0,Y 759.919,Z 853.739,A -85,B 0,C 180,E1 296.491,E2 296.491} C_VEL
LIN {X 0,Y 759.916,Z 875.252,A -85,B 0,C 180,E1 295.651,E2 295.651} C_VEL
LIN {X 0,Y 759.913,Z 894.66,A -85,B 0,C 180,E1 294.783,E2 294.783} C_VEL
LIN {X 0,Y 759.911,Z 917.061,A -85,B 0,C 180,E1 293.62,E2 293.62} C_VEL
LIN {X 0,Y 759.907,Z 935.706,A -85,B 0,C 180,E1 292.513,E2 292.513} C_VEL
LIN {X 0,Y 759.909,Z 955.524,A -85,B 0,C 180,E1 291.173,E2 291.173} C_VEL
LIN {X 0,Y 759.917,Z 972.885,A -85,B 0,C 180,E1 289.845,E2 289.845} C_VEL
LIN {X 0,Y 759.909,Z 989.391,A -85,B 0,C 180,E1 288.409,E2 288.409} C_VEL
LIN {X 0,Y 759.903,Z 1003.947,A -85,B 0,C 180,E1 286.984,E2 286.984} C_VEL
LIN {X 0,Y 759.915,Z 1018.836,A -85,B 0,C 180,E1 285.317,E2 285.317} C_VEL
LIN {X 0,Y 759.898,Z 1030.589,A -85,B 0,C 180,E1 283.812,E2 283.812} C_VEL
LIN {X 0,Y 759.901,Z 1042.785,A -85,B 0,C 180,E1 281.999,E2 281.999} C_VEL
LIN {X 0,Y 759.91,Z 1051.555,A -85,B 0,C 180,E1 280.462,E2 280.462} C_VEL
LIN {X 0,Y 759.89,Z 1060.073,A -85,B 0,C 180,E1 278.703,E2 278.703} C_VEL
LIN {X 0,Y 759.919,Z 1066.726,A -85,B 0,C 180,E1 276.953,E2 276.953} C_VEL
LIN {X 0,Y 759.906,Z 1071.51,A -85,B 0,C 180,E1 275.361,E2 275.361} C_VEL
LIN {X 0,Y 759.917,Z 1075.671,A -85,B 0,C 180,E1 273.395,E2 273.395} C_VEL
LIN {X 0,Y 759.899,Z 1077.63,A -85,B 0,C 180,E1 271.81,E2 271.81} C_VEL
LIN {X 0,Y 759.92,Z 1078.5,A -85,B 0,C 180,E1 270,E2 270} C_VEL
LIN {X 0,Y 759.899,Z 1077.63,A -85,B 0,C 180,E1 268.19,E2 268.19} C_VEL
LIN {X 0,Y 759.918,Z 1075.559,A -85,B 0,C 180,E1 266.53,E2 266.53} C_VEL
LIN {X 0,Y 759.906,Z 1071.51,A -85,B 0,C 180,E1 264.639,E2 264.639} C_VEL
LIN {X 0,Y 759.919,Z 1066.726,A -85,B 0,C 180,E1 263.047,E2 263.047} C_VEL
LIN {X 0,Y 759.892,Z 1059.729,A -85,B 0,C 180,E1 261.22,E2 261.22} C_VEL
LIN {X 0,Y 759.91,Z 1051.555,A -85,B 0,C 180,E1 259.538,E2 259.538} C_VEL
LIN {X 0,Y 759.901,Z 1042.786,A -85,B 0,C 180,E1 258.001,E2 258.001} C_VEL
LIN {X 0,Y 759.898,Z 1030.589,A -85,B 0,C 180,E1 256.188,E2 256.188} C_VEL
LIN {X 0,Y 759.917,Z 1018.833,A -85,B 0,C 180,E1 254.683,E2 254.683} C_VEL
LIN {X 0,Y 759.903,Z 1003.948,A -85,B 0,C 180,E1 253.016,E2 253.016} C_VEL
LIN {X 0,Y 759.909,Z 989.391,A -85,B 0,C 180,E1 251.591,E2 251.591} C_VEL
LIN {X 0,Y 759.911,Z 971.366,A -85,B 0,C 180,E1 250.035,E2 250.035} C_VEL
LIN {X 0,Y 759.913,Z 954.42,A -85,B 0,C 180,E1 248.746,E2 248.746} C_VEL
LIN {X 0,Y 759.909,Z 934.383,A -85,B 0,C 180,E1 247.405,E2 247.405} C_VEL
LIN {X 0,Y 759.91,Z 915.991,A -85,B 0,C 180,E1 246.32,E2 246.32} C_VEL
LIN {X 0,Y 759.912,Z 893.9,A -85,B 0,C 180,E1 245.182,E2 245.182} C_VEL
LIN {X 0,Y 759.916,Z 874.865,A -85,B 0,C 180,E1 244.332,E2 244.332} C_VEL
LIN {X 0,Y 759.916,Z 852.82,A -85,B 0,C 180,E1 243.475,E2 243.475} C_VEL
LIN {X 0,Y 759.901,Z 831.087,A -85,B 0,C 180,E1 242.779,E2 242.779} C_VEL
LIN {X 0,Y 759.902,Z 811.685,A -85,B 0,C 180,E1 242.258,E2 242.258} C_VEL
LIN {X 0,Y 759.899,Z 789.26,A -85,B 0,C 180,E1 241.768,E2 241.768} C_VEL
LIN {X 0,Y 759.917,Z 765.997,A -85,B 0,C 180,E1 241.405,E2 241.405} C_VEL
LIN {X 0,Y 759.899,Z 499.217,A -85,B 0,C 180,E1 238.53,E2 238.53} C_VEL
LIN {X 0,Y 759.911,Z 376.685,A -85,B 0,C 180,E1 237.173,E2 237.173} C_VEL
LIN {X 0,Y 759.853,Z 337.913,A -85,B 0,C 180,E1 234.582,E2 234.582} C_VEL
LIN {X 0,Y 759.861,Z 326.575,A -85,B 0,C 180,E1 233.784,E2 233.784} C_VEL
LIN {X 0,Y 759.887,Z 326.577,A -85,B 0,C 180,E1 230.808,E2 230.808} C_VEL
LIN {X 0,Y 759.841,Z 326.574,A -85,B 0,C 180,E1 228.252,E2 228.252} C_VEL
LIN {X 0,Y 759.85,Z 326.572,A -85,B 0,C 180,E1 225.779,E2 225.779} C_VEL
LIN {X 0,Y 759.913,Z 326.575,A -85,B 0,C 180,E1 222.968,E2 222.968} C_VEL
LIN {X 0,Y 759.847,Z 326.574,A -85,B 0,C 180,E1 220.249,E2 220.249} C_VEL
LIN {X 0,Y 759.841,Z 326.572,A -85,B 0,C 180,E1 217.823,E2 217.823} C_VEL
LIN {X 0,Y 759.9,Z 326.569,A -85,B 0,C 180,E1 215.193,E2 215.193} C_VEL
LIN {X 0,Y 759.862,Z 326.575,A -85,B 0,C 180,E1 212.293,E2 212.293} C_VEL
LIN {X 0,Y 759.84,Z 326.573,A -85,B 0,C 180,E1 209.83,E2 209.83} C_VEL
LIN {X 0,Y 759.863,Z 326.57,A -85,B 0,C 180,E1 207.338,E2 207.338} C_VEL
LIN {X 0,Y 759.884,Z 326.576,A -85,B 0,C 180,E1 204.322,E2 204.322} C_VEL
LIN {X 0,Y 759.841,Z 326.574,A -85,B 0,C 180,E1 201.783,E2 201.783} C_VEL
LIN {X 0,Y 759.853,Z 326.571,A -85,B 0,C 180,E1 199.287,E2 199.287} C_VEL
LIN {X 0,Y 759.912,Z 326.577,A -85,B 0,C 180,E1 196.355,E2 196.355} C_VEL
LIN {X 0,Y 759.844,Z 326.574,A -85,B 0,C 180,E1 193.702,E2 193.702} C_VEL
LIN {X 0,Y 759.85,Z 326.571,A -85,B 0,C 180,E1 191.23,E2 191.23} C_VEL
LIN {X 0,Y 759.916,Z 326.573,A -85,B 0,C 180,E1 188.398,E2 188.398} C_VEL
LIN {X 0,Y 759.85,Z 326.574,A -85,B 0,C 180,E1 185.664,E2 185.664} C_VEL
LIN {X 0,Y 759.846,Z 326.571,A -85,B 0,C 180,E1 183.168,E2 183.168} C_VEL
LIN {X 0,Y 759.918,Z 326.569,A -85,B 0,C 180,E1 180.452,E2 180.452} C_VEL
LIN {X 0,Y 759.855,Z 326.575,A -85,B 0,C 180,E1 177.587,E2 177.587} C_VEL
LIN {X 0,Y 759.843,Z 326.572,A -85,B 0,C 180,E1 177.169,E2 177.169} C_VEL
LIN {X 0,Y 758.856,Z 326.699,A -85,B 0,C 180,E1 176.588,E2 176.588} C_VEL
LIN {X 0,Y 752.444,Z 327.495,A -85,B 0,C 180,E1 174.962,E2 174.962} C_VEL
LIN {X 0,Y 751.957,Z 327.557,A -85,B 0,C 180,E1 174.539,E2 174.539} C_VEL
LIN {X 0,Y 751.926,Z 327.564,A -85,B 0,C 180,E1 171.589,E2 171.589} C_VEL
LIN {X 0,Y 751.905,Z 327.56,A -85,B 0,C 180,E1 169.038,E2 169.038} C_VEL
LIN {X 0,Y 751.96,Z 327.558,A -85,B 0,C 180,E1 166.387,E2 166.387} C_VEL
LIN {X 0,Y 751.928,Z 327.564,A -85,B 0,C 180,E1 163.467,E2 163.467} C_VEL
LIN {X 0,Y 751.906,Z 327.561,A -85,B 0,C 180,E1 160.905,E2 160.905} C_VEL
LIN {X 0,Y 751.965,Z 327.556,A -85,B 0,C 180,E1 158.223,E2 158.223} C_VEL
LIN {X 0,Y 751.923,Z 327.563,A -85,B 0,C 180,E1 155.263,E2 155.263} C_VEL
LIN {X 0,Y 751.906,Z 327.561,A -85,B 0,C 180,E1 152.777,E2 152.777} C_VEL
LIN {X 0,Y 751.965,Z 327.556,A -85,B 0,C 180,E1 150.09,E2 150.09} C_VEL
LIN {X 0,Y 751.925,Z 327.563,A -85,B 0,C 180,E1 147.143,E2 147.143} C_VEL
LIN {X 0,Y 751.908,Z 327.561,A -85,B 0,C 180,E1 144.604,E2 144.604} C_VEL
LIN {X 0,Y 751.967,Z 327.558,A -85,B 0,C 180,E1 141.904,E2 141.904} C_VEL
LIN {X 0,Y 751.928,Z 327.565,A -85,B 0,C 180,E1 139.036,E2 139.036} C_VEL
LIN {X 0,Y 751.908,Z 327.559,A -85,B 0,C 180,E1 136.461,E2 136.461} C_VEL
LIN {X 0,Y 751.978,Z 327.557,A -85,B 0,C 180,E1 133.744,E2 133.744} C_VEL
LIN {X 0,Y 751.924,Z 327.564,A -85,B 0,C 180,E1 130.83,E2 130.83} C_VEL
LIN {X 0,Y 751.909,Z 327.562,A -85,B 0,C 180,E1 128.293,E2 128.293} C_VEL
LIN {X 0,Y 751.977,Z 327.56,A -85,B 0,C 180,E1 125.526,E2 125.526} C_VEL
LIN {X 0,Y 751.918,Z 327.57,A -85,B 0,C 180,E1 122.631,E2 122.631} C_VEL
LIN {X 0,Y 752.019,Z 328.205,A -85,B 0,C 180,E1 122.544,E2 122.544} C_VEL
LIN {X 0,Y 752.673,Z 330.551,A -85,B 0,C 180,E1 122.339,E2 122.339} C_VEL
LIN {X 0,Y 752.738,Z 347.819,A -85,B 0,C 180,E1 121.104,E2 121.104} C_VEL
LIN {X 0,Y 753.146,Z 351.266,A -85,B 0,C 180,E1 121.045,E2 121.045} C_VEL
LIN {X 0,Y 752.991,Z 587.579,A -85,B 0,C 180,E1 118.455,E2 118.455} C_VEL
LIN {X 0,Y 752.881,Z 736.326,A -85,B 0,C 180,E1 116.838,E2 116.838} C_VEL
LIN {X 0,Y 752.803,Z 761.088,A -85,B 0,C 180,E1 116.439,E2 116.439} C_VEL
LIN {X 0,Y 752.755,Z 782.475,A -85,B 0,C 180,E1 115.964,E2 115.964} C_VEL
LIN {X 0,Y 752.692,Z 803.068,A -85,B 0,C 180,E1 115.401,E2 115.401} C_VEL
LIN {X 0,Y 752.615,Z 827.719,A -85,B 0,C 180,E1 114.572,E2 114.572} C_VEL
LIN {X 0,Y 752.542,Z 847.477,A -85,B 0,C 180,E1 113.782,E2 113.782} C_VEL
LIN {X 0,Y 752.439,Z 869.885,A -85,B 0,C 180,E1 112.745,E2 112.745} C_VEL
LIN {X 0,Y 752.362,Z 889.573,A -85,B 0,C 180,E1 111.682,E2 111.682} C_VEL
LIN {X 0,Y 752.278,Z 909.967,A -85,B 0,C 180,E1 110.437,E2 110.437} C_VEL
LIN {X 0,Y 752.196,Z 928.613,A -85,B 0,C 180,E1 109.127,E2 109.127} C_VEL
LIN {X 0,Y 752.118,Z 947.271,A -85,B 0,C 180,E1 107.644,E2 107.644} C_VEL
LIN {X 0,Y 752.085,Z 962.369,A -85,B 0,C 180,E1 106.281,E2 106.281} C_VEL
LIN {X 0,Y 752.024,Z 979.192,A -85,B 0,C 180,E1 104.554,E2 104.554} C_VEL
LIN {X 0,Y 751.98,Z 991.869,A -85,B 0,C 180,E1 103.064,E2 103.064} C_VEL
LIN {X 0,Y 751.955,Z 1005.115,A -85,B 0,C 180,E1 101.272,E2 101.272} C_VEL
LIN {X 0,Y 751.932,Z 1014.93,A -85,B 0,C 180,E1 99.723,E2 99.723} C_VEL
LIN {X 0,Y 751.918,Z 1024.578,A -85,B 0,C 180,E1 97.949,E2 97.949} C_VEL
LIN {X 0,Y 751.919,Z 1032.319,A -85,B 0,C 180,E1 96.183,E2 96.183} C_VEL
LIN {X 0,Y 751.904,Z 1038.071,A -85,B 0,C 180,E1 94.576,E2 94.576} C_VEL
LIN {X 0,Y 751.913,Z 1043.37,A -85,B 0,C 180,E1 92.591,E2 92.591} C_VEL
LIN {X 0,Y 751.915,Z 1046.253,A -85,B 0,C 180,E1 90.991,E2 90.991} C_VEL
LIN {X 0,Y 751.913,Z 1048.154,A -85,B 0,C 180,E1 89.162,E2 89.162} C_VEL
LIN {X 0,Y 751.891,Z 1048.347,A -85,B 0,C 180,E1 87.409,E2 87.409} C_VEL
LIN {X 0,Y 751.918,Z 1047.283,A -85,B 0,C 180,E1 85.729,E2 85.729} C_VEL
LIN {X 0,Y 751.917,Z 1044.403,A -85,B 0,C 180,E1 83.817,E2 83.817} C_VEL
LIN {X 0,Y 751.915,Z 1040.55,A -85,B 0,C 180,E1 82.18,E2 82.18} C_VEL
LIN {X 0,Y 751.898,Z 1034.799,A -85,B 0,C 180,E1 80.354,E2 80.354} C_VEL
LIN {X 0,Y 751.919,Z 1027.386,A -85,B 0,C 180,E1 78.572,E2 78.572} C_VEL
LIN {X 0,Y 751.925,Z 1019.21,A -85,B 0,C 180,E1 76.935,E2 76.935} C_VEL
LIN {X 0,Y 751.938,Z 1008.38,A -85,B 0,C 180,E1 75.129,E2 75.129} C_VEL
LIN {X 0,Y 751.978,Z 997.883,A -85,B 0,C 180,E1 73.627,E2 73.627} C_VEL
LIN {X 0,Y 752.007,Z 984.331,A -85,B 0,C 180,E1 71.932,E2 71.932} C_VEL
LIN {X 0,Y 752.051,Z 970.413,A -85,B 0,C 180,E1 70.425,E2 70.425} C_VEL
LIN {X 0,Y 752.111,Z 954.372,A -85,B 0,C 180,E1 68.883,E2 68.883} C_VEL
LIN {X 0,Y 752.167,Z 937.802,A -85,B 0,C 180,E1 67.49,E2 67.49} C_VEL
LIN {X 0,Y 752.241,Z 918.335,A -85,B 0,C 180,E1 66.041,E2 66.041} C_VEL
LIN {X 0,Y 752.312,Z 900.432,A -85,B 0,C 180,E1 64.872,E2 64.872} C_VEL
LIN {X 0,Y 752.417,Z 879.19,A -85,B 0,C 180,E1 63.65,E2 63.65} C_VEL
LIN {X 0,Y 752.488,Z 859.592,A -85,B 0,C 180,E1 62.671,E2 62.671} C_VEL
LIN {X 0,Y 752.59,Z 838.022,A -85,B 0,C 180,E1 61.729,E2 61.729} C_VEL
LIN {X 0,Y 752.643,Z 815.482,A -85,B 0,C 180,E1 60.907,E2 60.907} C_VEL
LIN {X 0,Y 752.723,Z 795.82,A -85,B 0,C 180,E1 60.299,E2 60.299} C_VEL
LIN {X 0,Y 752.788,Z 770.26,A -85,B 0,C 180,E1 59.661,E2 59.661} C_VEL
LIN {X 0,Y 752.848,Z 750.065,A -85,B 0,C 180,E1 59.278,E2 59.278} C_VEL
LIN {X 0,Y 752.884,Z 728.753,A -85,B 0,C 180,E1 58.976,E2 58.976} C_VEL
LIN {X 0,Y 753.089,Z 467.381,A -85,B 0,C 180,E1 56.147,E2 56.147} C_VEL
LIN {X 0,Y 752.941,Z 348.669,A -85,B 0,C 180,E1 54.825,E2 54.825} C_VEL
LIN {X 0,Y 752.669,Z 347.331,A -85,B 0,C 180,E1 54.786,E2 54.786} C_VEL
LIN {X 0,Y 752.503,Z 329.753,A -85,B 0,C 180,E1 53.504,E2 53.504} C_VEL
LIN {X 0,Y 751.916,Z 327.57,A -85,B 0,C 180,E1 53.309,E2 53.309} C_VEL
LIN {X 0,Y 751.975,Z 327.561,A -85,B 0,C 180,E1 50.438,E2 50.438} C_VEL
LIN {X 0,Y 751.909,Z 327.561,A -85,B 0,C 180,E1 47.678,E2 47.678} C_VEL
LIN {X 0,Y 751.917,Z 327.564,A -85,B 0,C 180,E1 45.136,E2 45.136} C_VEL
LIN {X 0,Y 751.976,Z 327.559,A -85,B 0,C 180,E1 42.285,E2 42.285} C_VEL
LIN {X 0,Y 751.908,Z 327.56,A -85,B 0,C 180,E1 39.531,E2 39.531} C_VEL
LIN {X 0,Y 751.914,Z 327.563,A -85,B 0,C 180,E1 37.042,E2 37.042} C_VEL
LIN {X 0,Y 751.977,Z 327.56,A -85,B 0,C 180,E1 34.202,E2 34.202} C_VEL
LIN {X 0,Y 751.909,Z 327.56,A -85,B 0,C 180,E1 31.419,E2 31.419} C_VEL
LIN {X 0,Y 751.911,Z 327.563,A -85,B 0,C 180,E1 28.95,E2 28.95} C_VEL
LIN {X 0,Y 751.978,Z 327.562,A -85,B 0,C 180,E1 26.164,E2 26.164} C_VEL
LIN {X 0,Y 751.913,Z 327.56,A -85,B 0,C 180,E1 23.346,E2 23.346} C_VEL
LIN {X 0,Y 751.907,Z 327.562,A -85,B 0,C 180,E1 20.879,E2 20.879} C_VEL
LIN {X 0,Y 751.976,Z 327.565,A -85,B 0,C 180,E1 18.128,E2 18.128} C_VEL
LIN {X 0,Y 751.915,Z 327.56,A -85,B 0,C 180,E1 15.266,E2 15.266} C_VEL
LIN {X 0,Y 751.906,Z 327.562,A -85,B 0,C 180,E1 12.753,E2 12.753} C_VEL
LIN {X 0,Y 751.976,Z 327.564,A -85,B 0,C 180,E1 9.954,E2 9.954} C_VEL
LIN {X 0,Y 751.913,Z 327.56,A -85,B 0,C 180,E1 7.104,E2 7.104} C_VEL
LIN {X 0,Y 751.905,Z 327.562,A -85,B 0,C 180,E1 4.653,E2 4.653} C_VEL
LIN {X 0,Y 751.973,Z 327.566,A -85,B 0,C 180,E1 1.905,E2 1.905} C_VEL
LIN {X 0,Y 751.917,Z 327.56,A -85,B 0,C 180,E1 -0.991,E2 -0.991} C_VEL
LIN {X 0,Y 751.905,Z 327.562,A -85,B 0,C 180,E1 -3.507,E2 -3.507} C_VEL
LIN {X 0,Y 751.976,Z 327.565,A -85,B 0,C 180,E1 -6.26,E2 -6.26} C_VEL
LIN {X 0,Y 751.917,Z 327.56,A -85,B 0,C 180,E1 -9.105,E2 -9.105} C_VEL
LIN {X 0,Y 751.903,Z 327.561,A -85,B 0,C 180,E1 -11.584,E2 -11.584} C_VEL
LIN {X 0,Y 751.959,Z 327.566,A -85,B 0,C 180,E1 -14.241,E2 -14.241} C_VEL
LIN {X 0,Y 751.924,Z 327.56,A -85,B 0,C 180,E1 -17.17,E2 -17.17} C_VEL
LIN {X 0,Y 751.901,Z 327.561,A -85,B 0,C 180,E1 -19.693,E2 -19.693} C_VEL
LIN {X 0,Y 751.954,Z 327.566,A -85,B 0,C 180,E1 -22.352,E2 -22.352} C_VEL
LIN {X 0,Y 751.926,Z 327.56,A -85,B 0,C 180,E1 -25.278,E2 -25.278} C_VEL
LIN {X 0,Y 751.902,Z 327.562,A -85,B 0,C 180,E1 -27.831,E2 -27.831} C_VEL
LIN {X 0,Y 751.947,Z 327.565,A -85,B 0,C 180,E1 -30.44,E2 -30.44} C_VEL
LIN {X 0,Y 751.927,Z 327.56,A -85,B 0,C 180,E1 -33.403,E2 -33.403} C_VEL
LIN {X 0,Y 751.901,Z 327.562,A -85,B 0,C 180,E1 -35.918,E2 -35.918} C_VEL
LIN {X 0,Y 751.933,Z 327.565,A -85,B 0,C 180,E1 -38.487,E2 -38.487} C_VEL
LIN {X 0,Y 751.929,Z 327.56,A -85,B 0,C 180,E1 -41.526,E2 -41.526} C_VEL
LIN {X 0,Y 751.901,Z 327.563,A -85,B 0,C 180,E1 -44.102,E2 -44.102} C_VEL
LIN {X 0,Y 751.939,Z 327.566,A -85,B 0,C 180,E1 -46.674,E2 -46.674} C_VEL
LIN {X 0,Y 751.931,Z 327.561,A -85,B 0,C 180,E1 -49.64,E2 -49.64} C_VEL
LIN {X 0,Y 751.9,Z 327.564,A -85,B 0,C 180,E1 -52.19,E2 -52.19} C_VEL
LIN {X 0,Y 751.972,Z 327.565,A -85,B 0,C 180,E1 -53.437,E2 -53.437} C_VEL
LIN {X 0,Y 752.813,Z 331.086,A -85,B 0,C 180,E1 -53.729,E2 -53.729} C_VEL
LIN {X 0,Y 752.744,Z 367.134,A -85,B 0,C 180,E1 -56.181,E2 -56.181} C_VEL
LIN {X 0,Y 752.801,Z 377.401,A -85,B 0,C 180,E1 -56.849,E2 -56.849} C_VEL
LIN {X 0,Y 753.182,Z 380.848,A -85,B 0,C 180,E1 -56.907,E2 -56.907} C_VEL
LIN {X 0,Y 752.979,Z 638.162,A -85,B 0,C 180,E1 -59.722,E2 -59.722} C_VEL
LIN {X 0,Y 752.879,Z 766.53,A -85,B 0,C 180,E1 -61.119,E2 -61.119} C_VEL
LIN {X 0,Y 752.8,Z 791.576,A -85,B 0,C 180,E1 -61.526,E2 -61.526} C_VEL
LIN {X 0,Y 752.755,Z 812.708,A -85,B 0,C 180,E1 -61.997,E2 -61.997} C_VEL
LIN {X 0,Y 752.693,Z 833.682,A -85,B 0,C 180,E1 -62.572,E2 -62.572} C_VEL
LIN {X 0,Y 752.614,Z 857.11,A -85,B 0,C 180,E1 -63.36,E2 -63.36} C_VEL
LIN {X 0,Y 752.546,Z 876.248,A -85,B 0,C 180,E1 -64.121,E2 -64.121} C_VEL
LIN {X 0,Y 752.469,Z 897.462,A -85,B 0,C 180,E1 -65.088,E2 -65.088} C_VEL
LIN {X 0,Y 752.363,Z 918.518,A -85,B 0,C 180,E1 -66.212,E2 -66.212} C_VEL
LIN {X 0,Y 752.292,Z 938.354,A -85,B 0,C 180,E1 -67.411,E2 -67.411} C_VEL
LIN {X 0,Y 752.2,Z 957.679,A -85,B 0,C 180,E1 -68.759,E2 -68.759} C_VEL
LIN {X 0,Y 752.131,Z 975.816,A -85,B 0,C 180,E1 -70.184,E2 -70.184} C_VEL
LIN {X 0,Y 752.084,Z 991.944,A -85,B 0,C 180,E1 -71.634,E2 -71.634} C_VEL
LIN {X 0,Y 752.018,Z 1007.676,A -85,B 0,C 180,E1 -73.23,E2 -73.23} C_VEL
LIN {X 0,Y 751.997,Z 1020.607,A -85,B 0,C 180,E1 -74.736,E2 -74.736} C_VEL
LIN {X 0,Y 751.967,Z 1033.325,A -85,B 0,C 180,E1 -76.413,E2 -76.413} C_VEL
LIN {X 0,Y 751.924,Z 1044.175,A -85,B 0,C 180,E1 -78.105,E2 -78.105} C_VEL
LIN {X 0,Y 751.931,Z 1052.78,A -85,B 0,C 180,E1 -79.658,E2 -79.658} C_VEL
LIN {X 0,Y 751.904,Z 1061.598,A -85,B 0,C 180,E1 -81.589,E2 -81.589} C_VEL
LIN {X 0,Y 751.906,Z 1067.489,A -85,B 0,C 180,E1 -83.203,E2 -83.203} C_VEL
LIN {X 0,Y 751.916,Z 1072.701,A -85,B 0,C 180,E1 -85.041,E2 -85.041} C_VEL
LIN {X 0,Y 751.916,Z 1076.121,A -85,B 0,C 180,E1 -86.875,E2 -86.875} C_VEL
LIN {X 0,Y 751.903,Z 1078.099,A -85,B 0,C 180,E1 -88.705,E2 -88.705} C_VEL
LIN {X 0,Y 751.891,Z 1078.351,A -85,B 0,C 180,E1 -90.533,E2 -90.533} C_VEL
LIN {X 0,Y 751.913,Z 1077.296,A -85,B 0,C 180,E1 -92.21,E2 -92.21} C_VEL
LIN {X 0,Y 751.91,Z 1074.343,A -85,B 0,C 180,E1 -94.168,E2 -94.168} C_VEL
LIN {X 0,Y 751.916,Z 1070.687,A -85,B 0,C 180,E1 -95.724,E2 -95.724} C_VEL
LIN {X 0,Y 751.897,Z 1064.936,A -85,B 0,C 180,E1 -97.565,E2 -97.565} C_VEL
LIN {X 0,Y 751.919,Z 1057.524,A -85,B 0,C 180,E1 -99.353,E2 -99.353} C_VEL
LIN {X 0,Y 751.924,Z 1049.516,A -85,B 0,C 180,E1 -100.962,E2 -100.962} C_VEL
LIN {X 0,Y 751.948,Z 1038.35,A -85,B 0,C 180,E1 -102.83,E2 -102.83} C_VEL
LIN {X 0,Y 751.97,Z 1027.951,A -85,B 0,C 180,E1 -104.319,E2 -104.319} C_VEL
LIN {X 0,Y 751.999,Z 1014.677,A -85,B 0,C 180,E1 -105.984,E2 -105.984} C_VEL
LIN {X 0,Y 752.053,Z 1000.842,A -85,B 0,C 180,E1 -107.486,E2 -107.486} C_VEL
LIN {X 0,Y 752.108,Z 984.651,A -85,B 0,C 180,E1 -109.048,E2 -109.048} C_VEL
LIN {X 0,Y 752.165,Z 967.82,A -85,B 0,C 180,E1 -110.464,E2 -110.464} C_VEL
LIN {X 0,Y 752.242,Z 948.443,A -85,B 0,C 180,E1 -111.906,E2 -111.906} C_VEL
LIN {X 0,Y 752.311,Z 930.417,A -85,B 0,C 180,E1 -113.084,E2 -113.084} C_VEL
LIN {X 0,Y 752.415,Z 908.748,A -85,B 0,C 180,E1 -114.328,E2 -114.328} C_VEL
LIN {X 0,Y 752.488,Z 889.454,A -85,B 0,C 180,E1 -115.29,E2 -115.29} C_VEL
LIN {X 0,Y 752.594,Z 867.166,A -85,B 0,C 180,E1 -116.259,E2 -116.259} C_VEL
LIN {X 0,Y 752.646,Z 846.235,A -85,B 0,C 180,E1 -117.023,E2 -117.023} C_VEL
LIN {X 0,Y 752.717,Z 827.025,A -85,B 0,C 180,E1 -117.621,E2 -117.621} C_VEL
LIN {X 0,Y 752.782,Z 802.762,A -85,B 0,C 180,E1 -118.242,E2 -118.242} C_VEL
LIN {X 0,Y 752.842,Z 781.048,A -85,B 0,C 180,E1 -118.661,E2 -118.661} C_VEL
LIN {X 0,Y 752.883,Z 760.645,A -85,B 0,C 180,E1 -118.955,E2 -118.955} C_VEL
LIN {X 0,Y 753.066,Z 501.507,A -85,B 0,C 180,E1 -121.764,E2 -121.764} C_VEL
LIN {X 0,Y 753.009,Z 378.268,A -85,B 0,C 180,E1 -123.131,E2 -123.131} C_VEL
LIN {X 0,Y 752.714,Z 376.593,A -85,B 0,C 180,E1 -123.188,E2 -123.188} C_VEL
LIN {X 0,Y 752.785,Z 339.845,A -85,B 0,C 180,E1 -125.669,E2 -125.669} C_VEL
LIN {X 0,Y 752.791,Z 330.294,A -85,B 0,C 180,E1 -126.327,E2 -126.327} C_VEL
LIN {X 0,Y 751.973,Z 327.564,A -85,B 0,C 180,E1 -126.569,E2 -126.569} C_VEL
LIN {X 0,Y 751.916,Z 327.567,A -85,B 0,C 180,E1 -129.467,E2 -129.467} C_VEL
LIN {X 0,Y 751.902,Z 327.563,A -85,B 0,C 180,E1 -131.982,E2 -131.982} C_VEL
LIN {X 0,Y 751.97,Z 327.559,A -85,B 0,C 180,E1 -134.701,E2 -134.701} C_VEL
LIN {X 0,Y 751.917,Z 327.564,A -85,B 0,C 180,E1 -137.607,E2 -137.607} C_VEL
LIN {X 0,Y 751.902,Z 327.561,A -85,B 0,C 180,E1 -140.112,E2 -140.112} C_VEL
LIN {X 0,Y 751.965,Z 327.558,A -85,B 0,C 180,E1 -142.796,E2 -142.796} C_VEL
LIN {X 0,Y 751.923,Z 327.564,A -85,B 0,C 180,E1 -145.679,E2 -145.679} C_VEL
LIN {X 0,Y 751.901,Z 327.562,A -85,B 0,C 180,E1 -148.223,E2 -148.223} C_VEL
LIN {X 0,Y 751.942,Z 327.559,A -85,B 0,C 180,E1 -150.79,E2 -150.79} C_VEL
LIN {X 0,Y 751.926,Z 327.564,A -85,B 0,C 180,E1 -153.801,E2 -153.801} C_VEL
LIN {X 0,Y 751.902,Z 327.561,A -85,B 0,C 180,E1 -156.321,E2 -156.321} C_VEL
LIN {X 0,Y 751.937,Z 327.559,A -85,B 0,C 180,E1 -158.877,E2 -158.877} C_VEL
LIN {X 0,Y 751.934,Z 327.565,A -85,B 0,C 180,E1 -161.871,E2 -161.871} C_VEL
LIN {X 0,Y 751.903,Z 327.562,A -85,B 0,C 180,E1 -164.418,E2 -164.418} C_VEL
LIN {X 0,Y 751.937,Z 327.558,A -85,B 0,C 180,E1 -167.013,E2 -167.013} C_VEL
LIN {X 0,Y 751.93,Z 327.563,A -85,B 0,C 180,E1 -170.045,E2 -170.045} C_VEL
LIN {X 0,Y 751.903,Z 327.562,A -85,B 0,C 180,E1 -172.589,E2 -172.589} C_VEL
LIN {X 0,Y 751.943,Z 327.558,A -85,B 0,C 180,E1 -175.194,E2 -175.194} C_VEL
LIN {X 0,Y 751.932,Z 327.565,A -85,B 0,C 180,E1 -178.171,E2 -178.171} C_VEL
LIN {X 0,Y 751.905,Z 327.56,A -85,B 0,C 180,E1 -180.686,E2 -180.686} C_VEL
LIN {X 0,Y 751.937,Z 327.559,A -85,B 0,C 180,E1 -183.278,E2 -183.278} C_VEL
LIN {X 0,Y 751.957,Z 327.557,A -85,B 0,C 180,E1 -185.461,E2 -185.461} C_VEL
LIN {X 0,Y 751.038,Z 327.682,A -85,B 0,C 180,E1 -186.048,E2 -186.048} C_VEL
LIN {X 0,Y 744.514,Z 328.502,A -85,B 0,C 180,E1 -187.733,E2 -187.733} C_VEL
LIN {X 0,Y 744.026,Z 328.555,A -85,B 0,C 180,E1 -188.117,E2 -188.117} C_VEL
LIN {X 0,Y 743.967,Z 328.549,A -85,B 0,C 180,E1 -190.767,E2 -190.767} C_VEL
LIN {X 0,Y 743.989,Z 328.548,A -85,B 0,C 180,E1 -193.366,E2 -193.366} C_VEL
LIN {X 0,Y 744.006,Z 328.553,A -85,B 0,C 180,E1 -196.393,E2 -196.393} C_VEL
LIN {X 0,Y 743.967,Z 328.551,A -85,B 0,C 180,E1 -198.981,E2 -198.981} C_VEL
LIN {X 0,Y 743.996,Z 328.546,A -85,B 0,C 180,E1 -201.564,E2 -201.564} C_VEL
LIN {X 0,Y 743.995,Z 328.552,A -85,B 0,C 180,E1 -204.622,E2 -204.622} C_VEL
LIN {X 0,Y 743.967,Z 328.551,A -85,B 0,C 180,E1 -207.191,E2 -207.191} C_VEL
LIN {X 0,Y 744.012,Z 328.545,A -85,B 0,C 180,E1 -209.818,E2 -209.818} C_VEL
LIN {X 0,Y 743.992,Z 328.552,A -85,B 0,C 180,E1 -212.794,E2 -212.794} C_VEL
LIN {X 0,Y 743.968,Z 328.551,A -85,B 0,C 180,E1 -215.333,E2 -215.333} C_VEL
LIN {X 0,Y 744.023,Z 328.547,A -85,B 0,C 180,E1 -218.045,E2 -218.045} C_VEL
LIN {X 0,Y 743.988,Z 328.554,A -85,B 0,C 180,E1 -220.985,E2 -220.985} C_VEL
LIN {X 0,Y 743.968,Z 328.547,A -85,B 0,C 180,E1 -223.482,E2 -223.482} C_VEL
LIN {X 0,Y 744.029,Z 328.546,A -85,B 0,C 180,E1 -226.203,E2 -226.203} C_VEL
LIN {X 0,Y 743.985,Z 328.554,A -85,B 0,C 180,E1 -229.17,E2 -229.17} C_VEL
LIN {X 0,Y 743.971,Z 328.551,A -85,B 0,C 180,E1 -231.715,E2 -231.715} C_VEL
LIN {X 0,Y 744.033,Z 328.549,A -85,B 0,C 180,E1 -234.416,E2 -234.416} C_VEL
LIN {X 0,Y 744.036,Z 328.75,A -85,B 0,C 180,E1 -237.071,E2 -237.071} C_VEL
LIN {X 0,Y 745.502,Z 334.227,A -85,B 0,C 180,E1 -237.555,E2 -237.555} C_VEL
LIN {X 0,Y 745.558,Z 347.88,A -85,B 0,C 180,E1 -238.535,E2 -238.535} C_VEL
LIN {X 0,Y 746.434,Z 352.248,A -85,B 0,C 180,E1 -238.629,E2 -238.629} C_VEL
LIN {X 0,Y 746.09,Z 588.531,A -85,B 0,C 180,E1 -241.243,E2 -241.243} C_VEL
LIN {X 0,Y 745.863,Z 736.508,A -85,B 0,C 180,E1 -242.866,E2 -242.866} C_VEL
LIN {X 0,Y 745.725,Z 761.666,A -85,B 0,C 180,E1 -243.278,E2 -243.278} C_VEL
LIN {X 0,Y 745.624,Z 783.079,A -85,B 0,C 180,E1 -243.76,E2 -243.76} C_VEL
LIN {X 0,Y 745.497,Z 805.058,A -85,B 0,C 180,E1 -244.371,E2 -244.371} C_VEL
LIN {X 0,Y 745.324,Z 828.364,A -85,B 0,C 180,E1 -245.171,E2 -245.171} C_VEL
LIN {X 0,Y 745.183,Z 848.052,A -85,B 0,C 180,E1 -245.969,E2 -245.969} C_VEL
LIN {X 0,Y 744.976,Z 870.727,A -85,B 0,C 180,E1 -247.034,E2 -247.034} C_VEL
LIN {X 0,Y 744.819,Z 890.713,A -85,B 0,C 180,E1 -248.128,E2 -248.128} C_VEL
LIN {X 0,Y 744.633,Z 911.764,A -85,B 0,C 180,E1 -249.443,E2 -249.443} C_VEL
LIN {X 0,Y 744.494,Z 929.48,A -85,B 0,C 180,E1 -250.708,E2 -250.708} C_VEL
LIN {X 0,Y 744.334,Z 948.584,A -85,B 0,C 180,E1 -252.257,E2 -252.257} C_VEL
LIN {X 0,Y 744.247,Z 964.191,A -85,B 0,C 180,E1 -253.693,E2 -253.693} C_VEL
LIN {X 0,Y 744.133,Z 979.904,A -85,B 0,C 180,E1 -255.345,E2 -255.345} C_VEL
LIN {X 0,Y 744.062,Z 992.692,A -85,B 0,C 180,E1 -256.873,E2 -256.873} C_VEL
LIN {X 0,Y 744.001,Z 1005.783,A -85,B 0,C 180,E1 -258.684,E2 -258.684} C_VEL
LIN {X 0,Y 743.962,Z 1015.065,A -85,B 0,C 180,E1 -260.172,E2 -260.172} C_VEL
LIN {X 0,Y 743.94,Z 1024.68,A -85,B 0,C 180,E1 -261.965,E2 -261.965} C_VEL
LIN {X 0,Y 743.92,Z 1032.406,A -85,B 0,C 180,E1 -263.75,E2 -263.75} C_VEL
LIN {X 0,Y 743.907,Z 1038.397,A -85,B 0,C 180,E1 -265.452,E2 -265.452} C_VEL
LIN {X 0,Y 743.913,Z 1043.416,A -85,B 0,C 180,E1 -267.381,E2 -267.381} C_VEL
LIN {X 0,Y 743.915,Z 1046.286,A -85,B 0,C 180,E1 -268.999,E2 -268.999} C_VEL
LIN {X 0,Y 743.914,Z 1048.183,A -85,B 0,C 180,E1 -270.924,E2 -270.924} C_VEL
LIN {X 0,Y 743.893,Z 1048.318,A -85,B 0,C 180,E1 -272.696,E2 -272.696} C_VEL
LIN {X 0,Y 743.904,Z 1047.129,A -85,B 0,C 180,E1 -274.471,E2 -274.471} C_VEL
LIN {X 0,Y 743.913,Z 1044.199,A -85,B 0,C 180,E1 -276.328,E2 -276.328} C_VEL
LIN {X 0,Y 743.921,Z 1040.349,A -85,B 0,C 180,E1 -277.958,E2 -277.958} C_VEL
LIN {X 0,Y 743.911,Z 1034.101,A -85,B 0,C 180,E1 -279.907,E2 -279.907} C_VEL
LIN {X 0,Y 743.924,Z 1027.283,A -85,B 0,C 180,E1 -281.553,E2 -281.553} C_VEL
LIN {X 0,Y 743.953,Z 1019.092,A -85,B 0,C 180,E1 -283.208,E2 -283.208} C_VEL
LIN {X 0,Y 743.985,Z 1008.229,A -85,B 0,C 180,E1 -285.034,E2 -285.034} C_VEL
LIN {X 0,Y 744.044,Z 997.713,A -85,B 0,C 180,E1 -286.553,E2 -286.553} C_VEL
LIN {X 0,Y 744.124,Z 983.591,A -85,B 0,C 180,E1 -288.326,E2 -288.326} C_VEL
LIN {X 0,Y 744.185,Z 970.183,A -85,B 0,C 180,E1 -289.791,E2 -289.791} C_VEL
LIN {X 0,Y 744.322,Z 953.329,A -85,B 0,C 180,E1 -291.416,E2 -291.416} C_VEL
LIN {X 0,Y 744.428,Z 936.984,A -85,B 0,C 180,E1 -292.799,E2 -292.799} C_VEL
LIN {X 0,Y 744.595,Z 917.363,A -85,B 0,C 180,E1 -294.262,E2 -294.262} C_VEL
LIN {X 0,Y 744.726,Z 899.367,A -85,B 0,C 180,E1 -295.445,E2 -295.445} C_VEL
LIN {X 0,Y 744.936,Z 877.899,A -85,B 0,C 180,E1 -296.678,E2 -296.678} C_VEL
LIN {X 0,Y 745.08,Z 858.16,A -85,B 0,C 180,E1 -297.667,E2 -297.667} C_VEL
LIN {X 0,Y 745.301,Z 833.955,A -85,B 0,C 180,E1 -298.704,E2 -298.704} C_VEL
LIN {X 0,Y 745.412,Z 813.434,A -85,B 0,C 180,E1 -299.447,E2 -299.447} C_VEL
LIN {X 0,Y 745.617,Z 789.81,A -85,B 0,C 180,E1 -300.16,E2 -300.16} C_VEL
LIN {X 0,Y 745.707,Z 767.455,A -85,B 0,C 180,E1 -300.691,E2 -300.691} C_VEL
LIN {X 0,Y 745.812,Z 746.729,A -85,B 0,C 180,E1 -301.075,E2 -301.075} C_VEL
LIN {X 0,Y 745.905,Z 715.938,A -85,B 0,C 180,E1 -301.467,E2 -301.467} C_VEL
LIN {X 0,Y 746.291,Z 462.088,A -85,B 0,C 180,E1 -304.236,E2 -304.236} C_VEL
LIN {X 0,Y 746.261,Z 350.498,A -85,B 0,C 180,E1 -305.489,E2 -305.489} C_VEL
LIN {X 0,Y 745.481,Z 347.33,A -85,B 0,C 180,E1 -305.576,E2 -305.576} C_VEL
LIN {X 0,Y 745.285,Z 332.822,A -85,B 0,C 180,E1 -306.65,E2 -306.65} C_VEL
LIN {X 0,Y 744.016,Z 328.557,A -85,B 0,C 180,E1 -307.062,E2 -307.062} C_VEL
LIN {X 0,Y 743.986,Z 328.55,A -85,B 0,C 180,E1 -310.073,E2 -310.073} C_VEL
LIN {X 0,Y 743.969,Z 328.553,A -85,B 0,C 180,E1 -312.639,E2 -312.639} C_VEL
LIN {X 0,Y 744.036,Z 328.555,A -85,B 0,C 180,E1 -315.344,E2 -315.344} C_VEL
LIN {X 0,Y 743.977,Z 328.548,A -85,B 0,C 180,E1 -318.297,E2 -318.297} C_VEL
LIN {X 0,Y 743.971,Z 328.551,A -85,B 0,C 180,E1 -320.849,E2 -320.849} C_VEL
LIN {X 0,Y 744.038,Z 328.547,A -85,B 0,C 180,E1 -323.655,E2 -323.655} C_VEL
LIN {X 0,Y 743.975,Z 328.549,A -85,B 0,C 180,E1 -326.47,E2 -326.47} C_VEL
LIN {X 0,Y 743.972,Z 328.551,A -85,B 0,C 180,E1 -329.019,E2 -329.019} C_VEL
LIN {X 0,Y 744.039,Z 328.55,A -85,B 0,C 180,E1 -331.855,E2 -331.855} C_VEL
LIN {X 0,Y 743.973,Z 328.548,A -85,B 0,C 180,E1 -334.613,E2 -334.613} C_VEL
LIN {X 0,Y 743.972,Z 328.552,A -85,B 0,C 180,E1 -337.144,E2 -337.144} C_VEL
LIN {X 0,Y 744.038,Z 328.551,A -85,B 0,C 180,E1 -339.959,E2 -339.959} C_VEL
LIN {X 0,Y 743.971,Z 328.549,A -85,B 0,C 180,E1 -342.802,E2 -342.802} C_VEL
LIN {X 0,Y 743.972,Z 328.552,A -85,B 0,C 180,E1 -345.285,E2 -345.285} C_VEL
LIN {X 0,Y 744.039,Z 328.55,A -85,B 0,C 180,E1 -348.135,E2 -348.135} C_VEL
LIN {X 0,Y 743.97,Z 328.549,A -85,B 0,C 180,E1 -350.953,E2 -350.953} C_VEL
LIN {X 0,Y 743.971,Z 328.552,A -85,B 0,C 180,E1 -353.44,E2 -353.44} C_VEL
LIN {X 0,Y 744.038,Z 328.55,A -85,B 0,C 180,E1 -356.301,E2 -356.301} C_VEL
LIN {X 0,Y 743.971,Z 328.549,A -85,B 0,C 180,E1 -359.076,E2 -359.076} C_VEL
LIN {X 0,Y 743.969,Z 328.552,A -85,B 0,C 180,E1 -361.54,E2 -361.54} C_VEL
LIN {X 0,Y 744.039,Z 328.551,A -85,B 0,C 180,E1 -364.393,E2 -364.393} C_VEL
LIN {X 0,Y 743.971,Z 328.548,A -85,B 0,C 180,E1 -367.18,E2 -367.18} C_VEL
LIN {X 0,Y 743.968,Z 328.552,A -85,B 0,C 180,E1 -369.672,E2 -369.672} C_VEL
LIN {X 0,Y 744.038,Z 328.552,A -85,B 0,C 180,E1 -372.496,E2 -372.496} C_VEL
LIN {X 0,Y 743.973,Z 328.548,A -85,B 0,C 180,E1 -375.273,E2 -375.273} C_VEL
LIN {X 0,Y 743.966,Z 328.552,A -85,B 0,C 180,E1 -377.764,E2 -377.764} C_VEL
LIN {X 0,Y 744.037,Z 328.554,A -85,B 0,C 180,E1 -380.533,E2 -380.533} C_VEL
LIN {X 0,Y 743.976,Z 328.548,A -85,B 0,C 180,E1 -383.373,E2 -383.373} C_VEL
LIN {X 0,Y 743.963,Z 328.552,A -85,B 0,C 180,E1 -385.815,E2 -385.815} C_VEL
LIN {X 0,Y 744.021,Z 328.554,A -85,B 0,C 180,E1 -388.495,E2 -388.495} C_VEL
LIN {X 0,Y 743.981,Z 328.549,A -85,B 0,C 180,E1 -391.431,E2 -391.431} C_VEL
LIN {X 0,Y 743.963,Z 328.552,A -85,B 0,C 180,E1 -393.901,E2 -393.901} C_VEL
LIN {X 0,Y 744.006,Z 328.555,A -85,B 0,C 180,E1 -396.539,E2 -396.539} C_VEL
LIN {X 0,Y 743.987,Z 328.549,A -85,B 0,C 180,E1 -399.517,E2 -399.517} C_VEL
LIN {X 0,Y 743.963,Z 328.551,A -85,B 0,C 180,E1 -402.014,E2 -402.014} C_VEL
LIN {X 0,Y 743.993,Z 328.554,A -85,B 0,C 180,E1 -404.578,E2 -404.578} C_VEL
LIN {X 0,Y 743.986,Z 328.55,A -85,B 0,C 180,E1 -407.662,E2 -407.662} C_VEL
LIN {X 0,Y 743.962,Z 328.553,A -85,B 0,C 180,E1 -410.127,E2 -410.127} C_VEL
LIN {X 0,Y 743.98,Z 328.556,A -85,B 0,C 180,E1 -412.593,E2 -412.593} C_VEL
LIN {X 0,Y 744.045,Z 328.588,A -85,B 0,C 180,E1 -413.056,E2 -413.056} C_VEL
LIN {X 0,Y 745.78,Z 334.387,A -85,B 0,C 180,E1 -413.563,E2 -413.563} C_VEL
LIN {X 0,Y 745.596,Z 369.862,A -85,B 0,C 180,E1 -415.998,E2 -415.998} C_VEL
LIN {X 0,Y 745.658,Z 377.522,A -85,B 0,C 180,E1 -416.492,E2 -416.492} C_VEL
LIN {X 0,Y 746.472,Z 381.703,A -85,B 0,C 180,E1 -416.58,E2 -416.58} C_VEL
LIN {X 0,Y 746.062,Z 639.18,A -85,B 0,C 180,E1 -419.423,E2 -419.423} C_VEL
LIN {X 0,Y 745.862,Z 766.637,A -85,B 0,C 180,E1 -420.823,E2 -420.823} C_VEL
LIN {X 0,Y 745.723,Z 791.762,A -85,B 0,C 180,E1 -421.235,E2 -421.235} C_VEL
LIN {X 0,Y 745.624,Z 813.142,A -85,B 0,C 180,E1 -421.716,E2 -421.716} C_VEL
LIN {X 0,Y 745.497,Z 835.888,A -85,B 0,C 180,E1 -422.35,E2 -422.35} C_VEL
LIN {X 0,Y 745.319,Z 859.238,A -85,B 0,C 180,E1 -423.16,E2 -423.16} C_VEL
LIN {X 0,Y 745.177,Z 879.235,A -85,B 0,C 180,E1 -423.974,E2 -423.974} C_VEL
LIN {X 0,Y 744.961,Z 902.334,A -85,B 0,C 180,E1 -425.074,E2 -425.074} C_VEL
LIN {X 0,Y 744.818,Z 921.356,A -85,B 0,C 180,E1 -426.12,E2 -426.12} C_VEL
LIN {X 0,Y 744.619,Z 943.232,A -85,B 0,C 180,E1 -427.499,E2 -427.499} C_VEL
LIN {X 0,Y 744.488,Z 960.818,A -85,B 0,C 180,E1 -428.762,E2 -428.762} C_VEL
LIN {X 0,Y 744.337,Z 978.603,A -85,B 0,C 180,E1 -430.213,E2 -430.213} C_VEL
LIN {X 0,Y 744.244,Z 994.496,A -85,B 0,C 180,E1 -431.677,E2 -431.677} C_VEL
LIN {X 0,Y 744.133,Z 1009.8,A -85,B 0,C 180,E1 -433.289,E2 -433.289} C_VEL
LIN {X 0,Y 744.067,Z 1023.175,A -85,B 0,C 180,E1 -434.888,E2 -434.888} C_VEL
LIN {X 0,Y 744.007,Z 1035.899,A -85,B 0,C 180,E1 -436.657,E2 -436.657} C_VEL
LIN {X 0,Y 743.953,Z 1045.564,A -85,B 0,C 180,E1 -438.212,E2 -438.212} C_VEL
LIN {X 0,Y 743.922,Z 1055.47,A -85,B 0,C 180,E1 -440.093,E2 -440.093} C_VEL
LIN {X 0,Y 743.921,Z 1062.51,A -85,B 0,C 180,E1 -441.731,E2 -441.731} C_VEL
LIN {X 0,Y 743.897,Z 1068.506,A -85,B 0,C 180,E1 -443.44,E2 -443.44} C_VEL
LIN {X 0,Y 743.916,Z 1073.495,A -85,B 0,C 180,E1 -445.374,E2 -445.374} C_VEL
LIN {X 0,Y 743.912,Z 1076.459,A -85,B 0,C 180,E1 -447.072,E2 -447.072} C_VEL
LIN {X 0,Y 743.91,Z 1078.24,A -85,B 0,C 180,E1 -449.076,E2 -449.076} C_VEL
LIN {X 0,Y 743.894,Z 1078.306,A -85,B 0,C 180,E1 -450.693,E2 -450.693} C_VEL
LIN {X 0,Y 743.906,Z 1077.017,A -85,B 0,C 180,E1 -452.542,E2 -452.542} C_VEL
LIN {X 0,Y 743.901,Z 1073.971,A -85,B 0,C 180,E1 -454.394,E2 -454.394} C_VEL
LIN {X 0,Y 743.913,Z 1070.069,A -85,B 0,C 180,E1 -456.018,E2 -456.018} C_VEL
LIN {X 0,Y 743.916,Z 1063.726,A -85,B 0,C 180,E1 -457.958,E2 -457.958} C_VEL
LIN {X 0,Y 743.917,Z 1056.89,A -85,B 0,C 180,E1 -459.594,E2 -459.594} C_VEL
LIN {X 0,Y 743.973,Z 1047.87,A -85,B 0,C 180,E1 -461.395,E2 -461.395} C_VEL
LIN {X 0,Y 743.998,Z 1037.312,A -85,B 0,C 180,E1 -463.128,E2 -463.128} C_VEL
LIN {X 0,Y 744.045,Z 1026.214,A -85,B 0,C 180,E1 -464.714,E2 -464.714} C_VEL
LIN {X 0,Y 744.124,Z 1012.63,A -85,B 0,C 180,E1 -466.39,E2 -466.39} C_VEL
LIN {X 0,Y 744.184,Z 999.29,A -85,B 0,C 180,E1 -467.839,E2 -467.839} C_VEL
LIN {X 0,Y 744.331,Z 982.319,A -85,B 0,C 180,E1 -469.46,E2 -469.46} C_VEL
LIN {X 0,Y 744.429,Z 966.464,A -85,B 0,C 180,E1 -470.797,E2 -470.797} C_VEL
LIN {X 0,Y 744.599,Z 946.854,A -85,B 0,C 180,E1 -472.252,E2 -472.252} C_VEL
LIN {X 0,Y 744.739,Z 928.435,A -85,B 0,C 180,E1 -473.458,E2 -473.458} C_VEL
LIN {X 0,Y 744.94,Z 906.546,A -85,B 0,C 180,E1 -474.705,E2 -474.705} C_VEL
LIN {X 0,Y 745.09,Z 886.788,A -85,B 0,C 180,E1 -475.687,E2 -475.687} C_VEL
LIN {X 0,Y 745.305,Z 863.326,A -85,B 0,C 180,E1 -476.683,E2 -476.683} C_VEL
LIN {X 0,Y 745.413,Z 843.693,A -85,B 0,C 180,E1 -477.393,E2 -477.393} C_VEL
LIN {X 0,Y 745.617,Z 820.256,A -85,B 0,C 180,E1 -478.104,E2 -478.104} C_VEL
LIN {X 0,Y 745.705,Z 797.576,A -85,B 0,C 180,E1 -478.644,E2 -478.644} C_VEL
LIN {X 0,Y 745.809,Z 776.999,A -85,B 0,C 180,E1 -479.026,E2 -479.026} C_VEL
LIN {X 0,Y 745.904,Z 746.257,A -85,B 0,C 180,E1 -479.418,E2 -479.418} C_VEL
LIN {X 0,Y 746.271,Z 496.106,A -85,B 0,C 180,E1 -482.147,E2 -482.147} C_VEL
LIN {X 0,Y 746.29,Z 379.921,A -85,B 0,C 180,E1 -483.449,E2 -483.449} C_VEL
LIN {X 0,Y 745.547,Z 376.685,A -85,B 0,C 180,E1 -483.542,E2 -483.542} C_VEL
LIN {X 0,Y 745.733,Z 341.21,A -85,B 0,C 180,E1 -485.964,E2 -485.964} C_VEL
LIN {X 0,Y 745.691,Z 333.581,A -85,B 0,C 180,E1 -486.499,E2 -486.499} C_VEL
LIN {X 0,Y 744.039,Z 328.555,A -85,B 0,C 180,E1 -486.969,E2 -486.969} C_VEL
LIN {X 0,Y 743.965,Z 328.556,A -85,B 0,C 180,E1 -489.673,E2 -489.673} C_VEL
LIN {X 0,Y 743.969,Z 328.552,A -85,B 0,C 180,E1 -492.117,E2 -492.117} C_VEL
LIN {X 0,Y 744.04,Z 328.553,A -85,B 0,C 180,E1 -494.981,E2 -494.981} C_VEL
LIN {X 0,Y 743.968,Z 328.553,A -85,B 0,C 180,E1 -497.778,E2 -497.778} C_VEL
LIN {X 0,Y 743.968,Z 328.549,A -85,B 0,C 180,E1 -500.243,E2 -500.243} C_VEL
LIN {X 0,Y 744.037,Z 328.549,A -85,B 0,C 180,E1 -502.983,E2 -502.983} C_VEL
LIN {X 0,Y 743.973,Z 328.552,A -85,B 0,C 180,E1 -505.82,E2 -505.82} C_VEL
LIN {X 0,Y 743.964,Z 328.55,A -85,B 0,C 180,E1 -508.298,E2 -508.298} C_VEL
LIN {X 0,Y 744.041,Z 328.548,A -85,B 0,C 180,E1 -511.067,E2 -511.067} C_VEL
LIN {X 0,Y 743.976,Z 328.553,A -85,B 0,C 180,E1 -513.929,E2 -513.929} C_VEL
LIN {X 0,Y 743.966,Z 328.549,A -85,B 0,C 180,E1 -516.435,E2 -516.435} C_VEL
LIN {X 0,Y 744.033,Z 328.547,A -85,B 0,C 180,E1 -519.137,E2 -519.137} C_VEL
LIN {X 0,Y 743.976,Z 328.553,A -85,B 0,C 180,E1 -522.075,E2 -522.075} C_VEL
LIN {X 0,Y 743.966,Z 328.55,A -85,B 0,C 180,E1 -524.567,E2 -524.567} C_VEL
LIN {X 0,Y 744.039,Z 328.547,A -85,B 0,C 180,E1 -527.347,E2 -527.347} C_VEL
LIN {X 0,Y 743.973,Z 328.55,A -85,B 0,C 180,E1 -530.25,E2 -530.25} C_VEL
LIN {X 0,Y 743.968,Z 328.55,A -85,B 0,C 180,E1 -532.742,E2 -532.742} C_VEL
LIN {X 0,Y 744.038,Z 328.548,A -85,B 0,C 180,E1 -535.53,E2 -535.53} C_VEL
LIN {X 0,Y 743.975,Z 328.552,A -85,B 0,C 180,E1 -538.383,E2 -538.383} C_VEL
LIN {X 0,Y 743.97,Z 328.547,A -85,B 0,C 180,E1 -540.924,E2 -540.924} C_VEL
LIN {X 0,Y 744.039,Z 328.551,A -85,B 0,C 180,E1 -543.776,E2 -543.776} C_VEL
LIN {X 0,Y 743.973,Z 328.551,A -85,B 0,C 180,E1 -546.56,E2 -546.56} C_VEL
LIN {X 0,Y 744.026,Z 328.555,A -85,B 0,C 180,E1 -548.117,E2 -548.117} C_VEL
LIN {X 0,Y 742.975,Z 328.677,A -85,B 0,C 180,E1 -548.711,E2 -548.711} C_VEL
LIN {X 0,Y 736.559,Z 329.479,A -85,B 0,C 180,E1 -550.372,E2 -550.372} C_VEL
LIN {X 0,Y 736.028,Z 329.537,A -85,B 0,C 180,E1 -550.804,E2 -550.804} C_VEL
LIN {X 0,Y 736.058,Z 329.537,A -85,B 0,C 180,E1 -553.433,E2 -553.433} C_VEL
LIN {X 0,Y 736.055,Z 329.542,A -85,B 0,C 180,E1 -556.494,E2 -556.494} C_VEL
LIN {X 0,Y 736.029,Z 329.539,A -85,B 0,C 180,E1 -559.111,E2 -559.111} C_VEL
LIN {X 0,Y 736.093,Z 329.534,A -85,B 0,C 180,E1 -561.851,E2 -561.851} C_VEL
LIN {X 0,Y 736.045,Z 329.539,A -85,B 0,C 180,E1 -564.734,E2 -564.734} C_VEL
LIN {X 0,Y 736.032,Z 329.539,A -85,B 0,C 180,E1 -567.321,E2 -567.321} C_VEL
LIN {X 0,Y 736.101,Z 329.534,A -85,B 0,C 180,E1 -570.086,E2 -570.086} C_VEL
LIN {X 0,Y 736.037,Z 329.539,A -85,B 0,C 180,E1 -573.008,E2 -573.008} C_VEL
LIN {X 0,Y 736.036,Z 329.538,A -85,B 0,C 180,E1 -575.551,E2 -575.551} C_VEL
LIN {X 0,Y 736.1,Z 329.542,A -85,B 0,C 180,E1 -578.472,E2 -578.472} C_VEL
LIN {X 0,Y 736.035,Z 329.542,A -85,B 0,C 180,E1 -581.214,E2 -581.214} C_VEL
LIN {X 0,Y 736.041,Z 329.534,A -85,B 0,C 180,E1 -583.746,E2 -583.746} C_VEL
LIN {X 0,Y 736.095,Z 329.545,A -85,B 0,C 180,E1 -586.688,E2 -586.688} C_VEL
LIN {X 0,Y 736.033,Z 329.542,A -85,B 0,C 180,E1 -589.411,E2 -589.411} C_VEL
LIN {X 0,Y 736.053,Z 329.539,A -85,B 0,C 180,E1 -592.021,E2 -592.021} C_VEL
LIN {X 0,Y 736.074,Z 329.545,A -85,B 0,C 180,E1 -595.023,E2 -595.023} C_VEL
LIN {X 0,Y 736.135,Z 329.792,A -85,B 0,C 180,E1 -596.719,E2 -596.719} C_VEL
LIN {X 0,Y 738.337,Z 337.129,A -85,B 0,C 180,E1 -597.389,E2 -597.389} C_VEL
LIN {X 0,Y 738.378,Z 347.878,A -85,B 0,C 180,E1 -598.166,E2 -598.166} C_VEL
LIN {X 0,Y 739.744,Z 353.96,A -85,B 0,C 180,E1 -598.306,E2 -598.306} C_VEL
LIN {X 0,Y 739.21,Z 590.191,A -85,B 0,C 180,E1 -600.943,E2 -600.943} C_VEL
LIN {X 0,Y 738.867,Z 736.606,A -85,B 0,C 180,E1 -602.564,E2 -602.564} C_VEL
LIN {X 0,Y 738.668,Z 761.853,A -85,B 0,C 180,E1 -602.981,E2 -602.981} C_VEL
LIN {X 0,Y 738.513,Z 783.409,A -85,B 0,C 180,E1 -603.471,E2 -603.471} C_VEL
LIN {X 0,Y 738.317,Z 806.613,A -85,B 0,C 180,E1 -604.125,E2 -604.125} C_VEL
LIN {X 0,Y 738.049,Z 829.01,A -85,B 0,C 180,E1 -604.91,E2 -604.91} C_VEL
LIN {X 0,Y 737.831,Z 849.605,A -85,B 0,C 180,E1 -605.756,E2 -605.756} C_VEL
LIN {X 0,Y 737.513,Z 872.31,A -85,B 0,C 180,E1 -606.848,E2 -606.848} C_VEL
LIN {X 0,Y 737.286,Z 891.854,A -85,B 0,C 180,E1 -607.935,E2 -607.935} C_VEL
LIN {X 0,Y 736.995,Z 913.308,A -85,B 0,C 180,E1 -609.303,E2 -609.303} C_VEL
LIN {X 0,Y 736.792,Z 931.058,A -85,B 0,C 180,E1 -610.593,E2 -610.593} C_VEL
LIN {X 0,Y 736.554,Z 949.348,A -85,B 0,C 180,E1 -612.107,E2 -612.107} C_VEL
LIN {X 0,Y 736.416,Z 965.272,A -85,B 0,C 180,E1 -613.595,E2 -613.595} C_VEL
LIN {X 0,Y 736.243,Z 980.534,A -85,B 0,C 180,E1 -615.233,E2 -615.233} C_VEL
LIN {X 0,Y 736.145,Z 993.512,A -85,B 0,C 180,E1 -616.809,E2 -616.809} C_VEL
LIN {X 0,Y 736.049,Z 1005.935,A -85,B 0,C 180,E1 -618.56,E2 -618.56} C_VEL
LIN {X 0,Y 735.993,Z 1015.659,A -85,B 0,C 180,E1 -620.144,E2 -620.144} C_VEL
LIN {X 0,Y 735.94,Z 1025.705,A -85,B 0,C 180,E1 -622.082,E2 -622.082} C_VEL
LIN {X 0,Y 735.923,Z 1032.494,A -85,B 0,C 180,E1 -623.682,E2 -623.682} C_VEL
LIN {X 0,Y 735.911,Z 1038.47,A -85,B 0,C 180,E1 -625.402,E2 -625.402} C_VEL
LIN {X 0,Y 735.911,Z 1043.461,A -85,B 0,C 180,E1 -627.352,E2 -627.352} C_VEL
LIN {X 0,Y 735.914,Z 1046.318,A -85,B 0,C 180,E1 -628.988,E2 -628.988} C_VEL
LIN {X 0,Y 735.914,Z 1048.189,A -85,B 0,C 180,E1 -630.934,E2 -630.934} C_VEL
LIN {X 0,Y 735.892,Z 1048.334,A -85,B 0,C 180,E1 -632.648,E2 -632.648} C_VEL
LIN {X 0,Y 735.912,Z 1047.245,A -85,B 0,C 180,E1 -634.364,E2 -634.364} C_VEL
LIN {X 0,Y 735.913,Z 1044.313,A -85,B 0,C 180,E1 -636.319,E2 -636.319} C_VEL
LIN {X 0,Y 735.923,Z 1040.497,A -85,B 0,C 180,E1 -637.966,E2 -637.966} C_VEL
LIN {X 0,Y 735.915,Z 1034.623,A -85,B 0,C 180,E1 -639.857,E2 -639.857} C_VEL
LIN {X 0,Y 735.935,Z 1027.538,A -85,B 0,C 180,E1 -641.6,E2 -641.6} C_VEL
LIN {X 0,Y 735.973,Z 1019.795,A -85,B 0,C 180,E1 -643.194,E2 -643.194} C_VEL
LIN {X 0,Y 736.032,Z 1008.602,A -85,B 0,C 180,E1 -645.119,E2 -645.119} C_VEL
LIN {X 0,Y 736.11,Z 998.128,A -85,B 0,C 180,E1 -646.655,E2 -646.655} C_VEL
LIN {X 0,Y 736.227,Z 984.804,A -85,B 0,C 180,E1 -648.366,E2 -648.366} C_VEL
LIN {X 0,Y 736.328,Z 970.74,A -85,B 0,C 180,E1 -649.928,E2 -649.928} C_VEL
LIN {X 0,Y 736.53,Z 954.755,A -85,B 0,C 180,E1 -651.503,E2 -651.503} C_VEL
LIN {X 0,Y 736.69,Z 938.221,A -85,B 0,C 180,E1 -652.926,E2 -652.926} C_VEL
LIN {X 0,Y 736.94,Z 919.455,A -85,B 0,C 180,E1 -654.36,E2 -654.36} C_VEL
LIN {X 0,Y 737.138,Z 901.371,A -85,B 0,C 180,E1 -655.572,E2 -655.572} C_VEL
LIN {X 0,Y 737.451,Z 880.688,A -85,B 0,C 180,E1 -656.797,E2 -656.797} C_VEL
LIN {X 0,Y 737.672,Z 860.35,A -85,B 0,C 180,E1 -657.837,E2 -657.837} C_VEL
LIN {X 0,Y 737.971,Z 838.881,A -85,B 0,C 180,E1 -658.795,E2 -658.795} C_VEL
LIN {X 0,Y 738.184,Z 815.929,A -85,B 0,C 180,E1 -659.653,E2 -659.653} C_VEL
LIN {X 0,Y 738.404,Z 794.836,A -85,B 0,C 180,E1 -660.315,E2 -660.315} C_VEL
LIN {X 0,Y 738.632,Z 769.892,A -85,B 0,C 180,E1 -660.939,E2 -660.939} C_VEL
LIN {X 0,Y 738.783,Z 749.231,A -85,B 0,C 180,E1 -661.335,E2 -661.335} C_VEL
LIN {X 0,Y 738.911,Z 725.248,A -85,B 0,C 180,E1 -661.671,E2 -661.671} C_VEL
LIN {X 0,Y 739.488,Z 471.878,A -85,B 0,C 180,E1 -664.458,E2 -664.458} C_VEL
LIN {X 0,Y 739.552,Z 352.325,A -85,B 0,C 180,E1 -665.812,E2 -665.812} C_VEL
LIN {X 0,Y 738.297,Z 347.255,A -85,B 0,C 180,E1 -665.951,E2 -665.951} C_VEL
LIN {X 0,Y 738.215,Z 336.227,A -85,B 0,C 180,E1 -666.775,E2 -666.775} C_VEL
LIN {X 0,Y 736.1,Z 329.543,A -85,B 0,C 180,E1 -667.411,E2 -667.411} C_VEL
LIN {X 0,Y 736.035,Z 329.541,A -85,B 0,C 180,E1 -670.229,E2 -670.229} C_VEL
LIN {X 0,Y 736.039,Z 329.544,A -85,B 0,C 180,E1 -672.813,E2 -672.813} C_VEL
LIN {X 0,Y 736.099,Z 329.536,A -85,B 0,C 180,E1 -675.717,E2 -675.717} C_VEL
LIN {X 0,Y 736.029,Z 329.538,A -85,B 0,C 180,E1 -678.475,E2 -678.475} C_VEL
LIN {X 0,Y 736.044,Z 329.541,A -85,B 0,C 180,E1 -681.026,E2 -681.026} C_VEL
LIN {X 0,Y 736.076,Z 329.53,A -85,B 0,C 180,E1 -684.058,E2 -684.058} C_VEL
LIN {X 0,Y 736.028,Z 329.54,A -85,B 0,C 180,E1 -686.713,E2 -686.713} C_VEL
LIN {X 0,Y 736.068,Z 329.542,A -85,B 0,C 180,E1 -689.375,E2 -689.375} C_VEL
LIN {X 0,Y 736.05,Z 329.538,A -85,B 0,C 180,E1 -692.404,E2 -692.404} C_VEL
LIN {X 0,Y 736.027,Z 329.539,A -85,B 0,C 180,E1 -694.974,E2 -694.974} C_VEL
LIN {X 0,Y 736.094,Z 329.543,A -85,B 0,C 180,E1 -697.729,E2 -697.729} C_VEL
LIN {X 0,Y 736.041,Z 329.538,A -85,B 0,C 180,E1 -700.642,E2 -700.642} C_VEL
LIN {X 0,Y 736.03,Z 329.54,A -85,B 0,C 180,E1 -703.18,E2 -703.18} C_VEL
LIN {X 0,Y 736.1,Z 329.54,A -85,B 0,C 180,E1 -706.008,E2 -706.008} C_VEL
LIN {X 0,Y 736.033,Z 329.538,A -85,B 0,C 180,E1 -708.878,E2 -708.878} C_VEL
LIN {X 0,Y 736.033,Z 329.541,A -85,B 0,C 180,E1 -711.406,E2 -711.406} C_VEL
LIN {X 0,Y 736.1,Z 329.538,A -85,B 0,C 180,E1 -714.231,E2 -714.231} C_VEL
LIN {X 0,Y 736.032,Z 329.539,A -85,B 0,C 180,E1 -717.041,E2 -717.041} C_VEL
LIN {X 0,Y 736.033,Z 329.54,A -85,B 0,C 180,E1 -719.533,E2 -719.533} C_VEL
LIN {X 0,Y 736.099,Z 329.538,A -85,B 0,C 180,E1 -722.336,E2 -722.336} C_VEL
LIN {X 0,Y 736.033,Z 329.539,A -85,B 0,C 180,E1 -725.144,E2 -725.144} C_VEL
LIN {X 0,Y 736.03,Z 329.539,A -85,B 0,C 180,E1 -727.651,E2 -727.651} C_VEL
LIN {X 0,Y 736.099,Z 329.537,A -85,B 0,C 180,E1 -730.488,E2 -730.488} C_VEL
LIN {X 0,Y 736.033,Z 329.539,A -85,B 0,C 180,E1 -733.273,E2 -733.273} C_VEL
LIN {X 0,Y 736.029,Z 329.539,A -85,B 0,C 180,E1 -735.765,E2 -735.765} C_VEL
LIN {X 0,Y 736.1,Z 329.537,A -85,B 0,C 180,E1 -738.616,E2 -738.616} C_VEL
LIN {X 0,Y 736.029,Z 329.539,A -85,B 0,C 180,E1 -741.477,E2 -741.477} C_VEL
LIN {X 0,Y 736.032,Z 329.539,A -85,B 0,C 180,E1 -743.966,E2 -743.966} C_VEL
LIN {X 0,Y 736.101,Z 329.538,A -85,B 0,C 180,E1 -746.818,E2 -746.818} C_VEL
LIN {X 0,Y 736.029,Z 329.539,A -85,B 0,C 180,E1 -749.607,E2 -749.607} C_VEL
LIN {X 0,Y 736.03,Z 329.542,A -85,B 0,C 180,E1 -752.085,E2 -752.085} C_VEL
LIN {X 0,Y 736.099,Z 329.541,A -85,B 0,C 180,E1 -754.881,E2 -754.881} C_VEL
LIN {X 0,Y 736.032,Z 329.539,A -85,B 0,C 180,E1 -757.685,E2 -757.685} C_VEL
LIN {X 0,Y 736.028,Z 329.542,A -85,B 0,C 180,E1 -760.187,E2 -760.187} C_VEL
LIN {X 0,Y 736.098,Z 329.542,A -85,B 0,C 180,E1 -762.993,E2 -762.993} C_VEL
LIN {X 0,Y 736.032,Z 329.54,A -85,B 0,C 180,E1 -765.831,E2 -765.831} C_VEL
LIN {X 0,Y 736.031,Z 329.543,A -85,B 0,C 180,E1 -768.371,E2 -768.371} C_VEL
LIN {X 0,Y 736.101,Z 329.543,A -85,B 0,C 180,E1 -771.233,E2 -771.233} C_VEL
LIN {X 0,Y 736.058,Z 329.629,A -85,B 0,C 180,E1 -772.661,E2 -772.661} C_VEL
LIN {X 0,Y 738.755,Z 337.51,A -85,B 0,C 180,E1 -773.381,E2 -773.381} C_VEL
LIN {X 0,Y 738.447,Z 373.273,A -85,B 0,C 180,E1 -775.858,E2 -775.858} C_VEL
LIN {X 0,Y 738.5,Z 377.442,A -85,B 0,C 180,E1 -776.122,E2 -776.122} C_VEL
LIN {X 0,Y 739.785,Z 383.425,A -85,B 0,C 180,E1 -776.257,E2 -776.257} C_VEL
LIN {X 0,Y 739.163,Z 641.852,A -85,B 0,C 180,E1 -779.136,E2 -779.136} C_VEL
LIN {X 0,Y 738.866,Z 766.745,A -85,B 0,C 180,E1 -780.521,E2 -780.521} C_VEL
LIN {X 0,Y 738.666,Z 792.02,A -85,B 0,C 180,E1 -780.939,E2 -780.939} C_VEL
LIN {X 0,Y 738.512,Z 813.469,A -85,B 0,C 180,E1 -781.427,E2 -781.427} C_VEL
LIN {X 0,Y 738.321,Z 836.62,A -85,B 0,C 180,E1 -782.08,E2 -782.08} C_VEL
LIN {X 0,Y 738.045,Z 859.542,A -85,B 0,C 180,E1 -782.885,E2 -782.885} C_VEL
LIN {X 0,Y 737.827,Z 880.233,A -85,B 0,C 180,E1 -783.739,E2 -783.739} C_VEL
LIN {X 0,Y 737.503,Z 903.14,A -85,B 0,C 180,E1 -784.847,E2 -784.847} C_VEL
LIN {X 0,Y 737.28,Z 922.886,A -85,B 0,C 180,E1 -785.95,E2 -785.95} C_VEL
LIN {X 0,Y 736.992,Z 943.234,A -85,B 0,C 180,E1 -787.253,E2 -787.253} C_VEL
LIN {X 0,Y 736.792,Z 961.106,A -85,B 0,C 180,E1 -788.551,E2 -788.551} C_VEL
LIN {X 0,Y 736.567,Z 978.603,A -85,B 0,C 180,E1 -789.996,E2 -789.996} C_VEL
LIN {X 0,Y 736.424,Z 994.494,A -85,B 0,C 180,E1 -791.475,E2 -791.475} C_VEL
LIN {X 0,Y 736.245,Z 1009.802,A -85,B 0,C 180,E1 -793.104,E2 -793.104} C_VEL
LIN {X 0,Y 736.159,Z 1022.669,A -85,B 0,C 180,E1 -794.658,E2 -794.658} C_VEL
LIN {X 0,Y 736.056,Z 1035.753,A -85,B 0,C 180,E1 -796.488,E2 -796.488} C_VEL
LIN {X 0,Y 735.988,Z 1045.128,A -85,B 0,C 180,E1 -798.007,E2 -798.007} C_VEL
LIN {X 0,Y 735.962,Z 1054.76,A -85,B 0,C 180,E1 -799.827,E2 -799.827} C_VEL
LIN {X 0,Y 735.918,Z 1062.206,A -85,B 0,C 180,E1 -801.562,E2 -801.562} C_VEL
LIN {X 0,Y 735.911,Z 1067.997,A -85,B 0,C 180,E1 -803.211,E2 -803.211} C_VEL
LIN {X 0,Y 735.917,Z 1073.178,A -85,B 0,C 180,E1 -805.168,E2 -805.168} C_VEL
LIN {X 0,Y 735.916,Z 1076.234,A -85,B 0,C 180,E1 -806.885,E2 -806.885} C_VEL
LIN {X 0,Y 735.907,Z 1078.149,A -85,B 0,C 180,E1 -808.754,E2 -808.754} C_VEL
LIN {X 0,Y 735.891,Z 1078.351,A -85,B 0,C 180,E1 -810.545,E2 -810.545} C_VEL
LIN {X 0,Y 735.914,Z 1077.297,A -85,B 0,C 180,E1 -812.258,E2 -812.258} C_VEL
LIN {X 0,Y 735.908,Z 1074.445,A -85,B 0,C 180,E1 -814.208,E2 -814.208} C_VEL
LIN {X 0,Y 735.918,Z 1070.688,A -85,B 0,C 180,E1 -815.849,E2 -815.849} C_VEL
LIN {X 0,Y 735.911,Z 1064.936,A -85,B 0,C 180,E1 -817.73,E2 -817.73} C_VEL
LIN {X 0,Y 735.931,Z 1057.601,A -85,B 0,C 180,E1 -819.541,E2 -819.541} C_VEL
LIN {X 0,Y 735.974,Z 1049.926,A -85,B 0,C 180,E1 -821.123,E2 -821.123} C_VEL
LIN {X 0,Y 736.039,Z 1038.526,A -85,B 0,C 180,E1 -823.086,E2 -823.086} C_VEL
LIN {X 0,Y 736.104,Z 1027.954,A -85,B 0,C 180,E1 -824.635,E2 -824.635} C_VEL
LIN {X 0,Y 736.23,Z 1014.045,A -85,B 0,C 180,E1 -826.409,E2 -826.409} C_VEL
LIN {X 0,Y 736.33,Z 1000.068,A -85,B 0,C 180,E1 -827.954,E2 -827.954} C_VEL
LIN {X 0,Y 736.542,Z 983.248,A -85,B 0,C 180,E1 -829.592,E2 -829.592} C_VEL
LIN {X 0,Y 736.708,Z 966.807,A -85,B 0,C 180,E1 -830.997,E2 -830.997} C_VEL
LIN {X 0,Y 736.965,Z 946.856,A -85,B 0,C 180,E1 -832.495,E2 -832.495} C_VEL
LIN {X 0,Y 737.196,Z 928.356,A -85,B 0,C 180,E1 -833.718,E2 -833.718} C_VEL
LIN {X 0,Y 737.48,Z 906.347,A -85,B 0,C 180,E1 -834.982,E2 -834.982} C_VEL
LIN {X 0,Y 737.719,Z 886.789,A -85,B 0,C 180,E1 -835.963,E2 -835.963} C_VEL
LIN {X 0,Y 738.022,Z 863.387,A -85,B 0,C 180,E1 -836.966,E2 -836.966} C_VEL
LIN {X 0,Y 738.198,Z 843.697,A -85,B 0,C 180,E1 -837.684,E2 -837.684} C_VEL
LIN {X 0,Y 738.494,Z 820.044,A -85,B 0,C 180,E1 -838.405,E2 -838.405} C_VEL
LIN {X 0,Y 738.641,Z 797.319,A -85,B 0,C 180,E1 -838.949,E2 -838.949} C_VEL
LIN {X 0,Y 738.792,Z 776.074,A -85,B 0,C 180,E1 -839.344,E2 -839.344} C_VEL
LIN {X 0,Y 738.933,Z 744.92,A -85,B 0,C 180,E1 -839.738,E2 -839.738} C_VEL
LIN {X 0,Y 739.5,Z 493.491,A -85,B 0,C 180,E1 -842.507,E2 -842.507} C_VEL
LIN {X 0,Y 739.604,Z 381.804,A -85,B 0,C 180,E1 -843.771,E2 -843.771} C_VEL
LIN {X 0,Y 738.409,Z 376.685,A -85,B 0,C 180,E1 -843.91,E2 -843.91} C_VEL
LIN {X 0,Y 738.712,Z 341.298,A -85,B 0,C 180,E1 -846.354,E2 -846.354} C_VEL
LIN {X 0,Y 738.481,Z 336.305,A -85,B 0,C 180,E1 -846.72,E2 -846.72} C_VEL
LIN {X 0,Y 736.045,Z 329.548,A -85,B 0,C 180,E1 -847.373,E2 -847.373} C_VEL
LIN {X 0,Y 736.024,Z 329.546,A -85,B 0,C 180,E1 -849.882,E2 -849.882} C_VEL
LIN {X 0,Y 736.063,Z 329.539,A -85,B 0,C 180,E1 -852.47,E2 -852.47} C_VEL
LIN {X 0,Y 736.046,Z 329.544,A -85,B 0,C 180,E1 -855.495,E2 -855.495} C_VEL
LIN {X 0,Y 736.024,Z 329.541,A -85,B 0,C 180,E1 -858.057,E2 -858.057} C_VEL
LIN {X 0,Y 736.082,Z 329.536,A -85,B 0,C 180,E1 -860.74,E2 -860.74} C_VEL
LIN {X 0,Y 736.042,Z 329.543,A -85,B 0,C 180,E1 -863.68,E2 -863.68} C_VEL
LIN {X 0,Y 736.026,Z 329.539,A -85,B 0,C 180,E1 -866.246,E2 -866.246} C_VEL
LIN {X 0,Y 736.099,Z 329.536,A -85,B 0,C 180,E1 -869.014,E2 -869.014} C_VEL
LIN {X 0,Y 736.038,Z 329.54,A -85,B 0,C 180,E1 -871.875,E2 -871.875} C_VEL
LIN {X 0,Y 736.028,Z 329.539,A -85,B 0,C 180,E1 -874.405,E2 -874.405} C_VEL
LIN {X 0,Y 736.1,Z 329.534,A -85,B 0,C 180,E1 -877.139,E2 -877.139} C_VEL
LIN {X 0,Y 736.034,Z 329.54,A -85,B 0,C 180,E1 -880.063,E2 -880.063} C_VEL
LIN {X 0,Y 736.031,Z 329.539,A -85,B 0,C 180,E1 -882.61,E2 -882.61} C_VEL
LIN {X 0,Y 736.099,Z 329.539,A -85,B 0,C 180,E1 -885.446,E2 -885.446} C_VEL
LIN {X 0,Y 736.033,Z 329.541,A -85,B 0,C 180,E1 -888.242,E2 -888.242} C_VEL
LIN {X 0,Y 736.033,Z 329.536,A -85,B 0,C 180,E1 -890.776,E2 -890.776} C_VEL
LIN {X 0,Y 736.1,Z 329.54,A -85,B 0,C 180,E1 -893.605,E2 -893.605} C_VEL
LIN {X 0,Y 736.032,Z 329.54,A -85,B 0,C 180,E1 -896.417,E2 -896.417} C_VEL
LIN {X 0,Y 736.037,Z 329.538,A -85,B 0,C 180,E1 -898.971,E2 -898.971} C_VEL
LIN {X 0,Y 736.097,Z 329.54,A -85,B 0,C 180,E1 -901.868,E2 -901.868} C_VEL
LIN {X 0,Y 736.03,Z 329.54,A -85,B 0,C 180,E1 -904.597,E2 -904.597} C_VEL
LIN {X 0,Y 736.037,Z 329.537,A -85,B 0,C 180,E1 -907.101,E2 -907.101} C_VEL
LIN {X 0,Y 736.097,Z 329.543,A -85,B 0,C 180,E1 -910.013,E2 -910.013} C_VEL
LIN {X 0,Y 736.028,Z 329.537,A -85,B 0,C 180,E1 -910.804,E2 -910.804} C_VEL
LIN {X 0,Y 735.028,Z 329.666,A -85,B 0,C 180,E1 -911.403,E2 -911.403} C_VEL
LIN {X 0,Y 728.625,Z 330.464,A -85,B 0,C 180,E1 -913.083,E2 -913.083} C_VEL
LIN {X 0,Y 728.13,Z 330.525,A -85,B 0,C 180,E1 -913.519,E2 -913.519} C_VEL
LIN {X 0,Y 728.109,Z 330.53,A -85,B 0,C 180,E1 -916.556,E2 -916.556} C_VEL
LIN {X 0,Y 728.092,Z 330.528,A -85,B 0,C 180,E1 -919.161,E2 -919.161} C_VEL
LIN {X 0,Y 728.159,Z 330.523,A -85,B 0,C 180,E1 -921.932,E2 -921.932} C_VEL
LIN {X 0,Y 728.097,Z 330.527,A -85,B 0,C 180,E1 -924.849,E2 -924.849} C_VEL
LIN {X 0,Y 728.096,Z 330.528,A -85,B 0,C 180,E1 -927.391,E2 -927.391} C_VEL
LIN {X 0,Y 728.16,Z 330.527,A -85,B 0,C 180,E1 -930.262,E2 -930.262} C_VEL
LIN {X 0,Y 728.093,Z 330.527,A -85,B 0,C 180,E1 -933.101,E2 -933.101} C_VEL
LIN {X 0,Y 728.11,Z 330.527,A -85,B 0,C 180,E1 -935.707,E2 -935.707} C_VEL
LIN {X 0,Y 728.13,Z 330.532,A -85,B 0,C 180,E1 -938.77,E2 -938.77} C_VEL
LIN {X 0,Y 728.092,Z 330.53,A -85,B 0,C 180,E1 -941.448,E2 -941.448} C_VEL
LIN {X 0,Y 728.156,Z 330.519,A -85,B 0,C 180,E1 -944.233,E2 -944.233} C_VEL
LIN {X 0,Y 728.104,Z 330.53,A -85,B 0,C 180,E1 -947.174,E2 -947.174} C_VEL
LIN {X 0,Y 728.099,Z 330.529,A -85,B 0,C 180,E1 -949.778,E2 -949.778} C_VEL
LIN {X 0,Y 728.161,Z 330.532,A -85,B 0,C 180,E1 -952.662,E2 -952.662} C_VEL
LIN {X 0,Y 728.095,Z 330.536,A -85,B 0,C 180,E1 -955.485,E2 -955.485} C_VEL
LIN {X 0,Y 728.157,Z 330.634,A -85,B 0,C 180,E1 -956.337,E2 -956.337} C_VEL
LIN {X 0,Y 731.175,Z 340.419,A -85,B 0,C 180,E1 -957.248,E2 -957.248} C_VEL
LIN {X 0,Y 731.211,Z 347.847,A -85,B 0,C 180,E1 -957.788,E2 -957.788} C_VEL
LIN {X 0,Y 733.078,Z 355.743,A -85,B 0,C 180,E1 -957.978,E2 -957.978} C_VEL
LIN {X 0,Y 732.35,Z 591.479,A -85,B 0,C 180,E1 -960.633,E2 -960.633} C_VEL
LIN {X 0,Y 731.891,Z 736.674,A -85,B 0,C 180,E1 -962.256,E2 -962.256} C_VEL
LIN {X 0,Y 731.635,Z 762.056,A -85,B 0,C 180,E1 -962.679,E2 -962.679} C_VEL
LIN {X 0,Y 731.419,Z 783.723,A -85,B 0,C 180,E1 -963.176,E2 -963.176} C_VEL
LIN {X 0,Y 731.163,Z 806.722,A -85,B 0,C 180,E1 -963.83,E2 -963.83} C_VEL
LIN {X 0,Y 730.791,Z 829.655,A -85,B 0,C 180,E1 -964.643,E2 -964.643} C_VEL
LIN {X 0,Y 730.482,Z 852.136,A -85,B 0,C 180,E1 -965.583,E2 -965.583} C_VEL
LIN {X 0,Y 730.067,Z 873.566,A -85,B 0,C 180,E1 -966.641,E2 -966.641} C_VEL
LIN {X 0,Y 729.754,Z 893.71,A -85,B 0,C 180,E1 -967.78,E2 -967.78} C_VEL
LIN {X 0,Y 729.388,Z 913.66,A -85,B 0,C 180,E1 -969.077,E2 -969.077} C_VEL
LIN {X 0,Y 729.096,Z 932.306,A -85,B 0,C 180,E1 -970.45,E2 -970.45} C_VEL
LIN {X 0,Y 728.785,Z 949.92,A -85,B 0,C 180,E1 -971.937,E2 -971.937} C_VEL
LIN {X 0,Y 728.585,Z 966.339,A -85,B 0,C 180,E1 -973.496,E2 -973.496} C_VEL
LIN {X 0,Y 728.356,Z 981.216,A -85,B 0,C 180,E1 -975.125,E2 -975.125} C_VEL
LIN {X 0,Y 728.216,Z 994.942,A -85,B 0,C 180,E1 -976.825,E2 -976.825} C_VEL
LIN {X 0,Y 728.096,Z 1006.602,A -85,B 0,C 180,E1 -978.514,E2 -978.514} C_VEL
LIN {X 0,Y 728.022,Z 1016.711,A -85,B 0,C 180,E1 -980.194,E2 -980.194} C_VEL
LIN {X 0,Y 727.951,Z 1026.298,A -85,B 0,C 180,E1 -982.105,E2 -982.105} C_VEL
LIN {X 0,Y 727.932,Z 1032.884,A -85,B 0,C 180,E1 -983.691,E2 -983.691} C_VEL
LIN {X 0,Y 727.913,Z 1039.273,A -85,B 0,C 180,E1 -985.588,E2 -985.588} C_VEL
LIN {X 0,Y 727.914,Z 1043.665,A -85,B 0,C 180,E1 -987.402,E2 -987.402} C_VEL
LIN {X 0,Y 727.906,Z 1046.575,A -85,B 0,C 180,E1 -989.134,E2 -989.134} C_VEL
LIN {X 0,Y 727.904,Z 1048.262,A -85,B 0,C 180,E1 -991.181,E2 -991.181} C_VEL
LIN {X 0,Y 727.9,Z 1048.283,A -85,B 0,C 180,E1 -992.835,E2 -992.835} C_VEL
LIN {X 0,Y 727.897,Z 1046.788,A -85,B 0,C 180,E1 -994.807,E2 -994.807} C_VEL
LIN {X 0,Y 727.916,Z 1043.949,A -85,B 0,C 180,E1 -996.547,E2 -996.547} C_VEL
LIN {X 0,Y 727.917,Z 1039.818,A -85,B 0,C 180,E1 -998.293,E2 -998.293} C_VEL
LIN {X 0,Y 727.938,Z 1033.314,A -85,B 0,C 180,E1 -1000.286,E2 -1000.286} C_VEL
LIN {X 0,Y 727.949,Z 1026.72,A -85,B 0,C 180,E1 -1001.89,E2 -1001.89} C_VEL
LIN {X 0,Y 728.024,Z 1018.026,A -85,B 0,C 180,E1 -1003.664,E2 -1003.664} C_VEL
LIN {X 0,Y 728.091,Z 1007.401,A -85,B 0,C 180,E1 -1005.451,E2 -1005.451} C_VEL
LIN {X 0,Y 728.196,Z 995.974,A -85,B 0,C 180,E1 -1007.121,E2 -1007.121} C_VEL
LIN {X 0,Y 728.355,Z 982.459,A -85,B 0,C 180,E1 -1008.821,E2 -1008.821} C_VEL
LIN {X 0,Y 728.531,Z 968.364,A -85,B 0,C 180,E1 -1010.38,E2 -1010.38} C_VEL
LIN {X 0,Y 728.763,Z 951.659,A -85,B 0,C 180,E1 -1011.998,E2 -1011.998} C_VEL
LIN {X 0,Y 729.047,Z 934.836,A -85,B 0,C 180,E1 -1013.437,E2 -1013.437} C_VEL
LIN {X 0,Y 729.341,Z 916.302,A -85,B 0,C 180,E1 -1014.828,E2 -1014.828} C_VEL
LIN {X 0,Y 729.671,Z 898.222,A -85,B 0,C 180,E1 -1016.031,E2 -1016.031} C_VEL
LIN {X 0,Y 730.026,Z 877.05,A -85,B 0,C 180,E1 -1017.262,E2 -1017.262} C_VEL
LIN {X 0,Y 730.364,Z 857.102,A -85,B 0,C 180,E1 -1018.274,E2 -1018.274} C_VEL
LIN {X 0,Y 730.753,Z 833.775,A -85,B 0,C 180,E1 -1019.286,E2 -1019.286} C_VEL
LIN {X 0,Y 731.015,Z 812.586,A -85,B 0,C 180,E1 -1020.064,E2 -1020.064} C_VEL
LIN {X 0,Y 731.403,Z 787.347,A -85,B 0,C 180,E1 -1020.821,E2 -1020.821} C_VEL
LIN {X 0,Y 731.608,Z 765.993,A -85,B 0,C 180,E1 -1021.328,E2 -1021.328} C_VEL
LIN {X 0,Y 731.866,Z 742.201,A -85,B 0,C 180,E1 -1021.761,E2 -1021.761} C_VEL
LIN {X 0,Y 732.018,Z 702.478,A -85,B 0,C 180,E1 -1022.231,E2 -1022.231} C_VEL
LIN {X 0,Y 732.808,Z 447.857,A -85,B 0,C 180,E1 -1025.065,E2 -1025.065} C_VEL
LIN {X 0,Y 732.898,Z 354.153,A -85,B 0,C 180,E1 -1026.14,E2 -1026.14} C_VEL
LIN {X 0,Y 731.135,Z 347.503,A -85,B 0,C 180,E1 -1026.311,E2 -1026.311} C_VEL
LIN {X 0,Y 731.178,Z 339.723,A -85,B 0,C 180,E1 -1026.894,E2 -1026.894} C_VEL
LIN {X 0,Y 728.14,Z 330.532,A -85,B 0,C 180,E1 -1027.767,E2 -1027.767} C_VEL
LIN {X 0,Y 728.09,Z 330.532,A -85,B 0,C 180,E1 -1030.464,E2 -1030.464} C_VEL
LIN {X 0,Y 728.135,Z 330.533,A -85,B 0,C 180,E1 -1033.146,E2 -1033.146} C_VEL
LIN {X 0,Y 728.111,Z 330.526,A -85,B 0,C 180,E1 -1036.134,E2 -1036.134} C_VEL
LIN {X 0,Y 728.09,Z 330.528,A -85,B 0,C 180,E1 -1038.694,E2 -1038.694} C_VEL
LIN {X 0,Y 728.154,Z 330.532,A -85,B 0,C 180,E1 -1041.433,E2 -1041.433} C_VEL
LIN {X 0,Y 728.101,Z 330.52,A -85,B 0,C 180,E1 -1044.389,E2 -1044.389} C_VEL
LIN {X 0,Y 728.094,Z 330.53,A -85,B 0,C 180,E1 -1046.962,E2 -1046.962} C_VEL
LIN {X 0,Y 728.161,Z 330.528,A -85,B 0,C 180,E1 -1049.829,E2 -1049.829} C_VEL
LIN {X 0,Y 728.096,Z 330.528,A -85,B 0,C 180,E1 -1052.609,E2 -1052.609} C_VEL
LIN {X 0,Y 728.098,Z 330.529,A -85,B 0,C 180,E1 -1055.195,E2 -1055.195} C_VEL
LIN {X 0,Y 728.153,Z 330.523,A -85,B 0,C 180,E1 -1058.167,E2 -1058.167} C_VEL
LIN {X 0,Y 728.089,Z 330.529,A -85,B 0,C 180,E1 -1060.922,E2 -1060.922} C_VEL
LIN {X 0,Y 728.121,Z 330.531,A -85,B 0,C 180,E1 -1063.567,E2 -1063.567} C_VEL
LIN {X 0,Y 728.117,Z 330.525,A -85,B 0,C 180,E1 -1066.58,E2 -1066.58} C_VEL
LIN {X 0,Y 728.089,Z 330.529,A -85,B 0,C 180,E1 -1069.155,E2 -1069.155} C_VEL
LIN {X 0,Y 728.149,Z 330.532,A -85,B 0,C 180,E1 -1071.92,E2 -1071.92} C_VEL
LIN {X 0,Y 728.101,Z 330.526,A -85,B 0,C 180,E1 -1074.879,E2 -1074.879} C_VEL
LIN {X 0,Y 728.089,Z 330.53,A -85,B 0,C 180,E1 -1077.402,E2 -1077.402} C_VEL
LIN {X 0,Y 728.163,Z 330.531,A -85,B 0,C 180,E1 -1080.236,E2 -1080.236} C_VEL
LIN {X 0,Y 728.097,Z 330.525,A -85,B 0,C 180,E1 -1083.07,E2 -1083.07} C_VEL
LIN {X 0,Y 728.091,Z 330.53,A -85,B 0,C 180,E1 -1085.596,E2 -1085.596} C_VEL
LIN {X 0,Y 728.162,Z 330.531,A -85,B 0,C 180,E1 -1088.37,E2 -1088.37} C_VEL
LIN {X 0,Y 728.094,Z 330.525,A -85,B 0,C 180,E1 -1091.245,E2 -1091.245} C_VEL
LIN {X 0,Y 728.091,Z 330.53,A -85,B 0,C 180,E1 -1093.744,E2 -1093.744} C_VEL
LIN {X 0,Y 728.16,Z 330.529,A -85,B 0,C 180,E1 -1096.596,E2 -1096.596} C_VEL
LIN {X 0,Y 728.09,Z 330.525,A -85,B 0,C 180,E1 -1099.411,E2 -1099.411} C_VEL
LIN {X 0,Y 728.093,Z 330.531,A -85,B 0,C 180,E1 -1101.934,E2 -1101.934} C_VEL
LIN {X 0,Y 728.162,Z 330.527,A -85,B 0,C 180,E1 -1104.815,E2 -1104.815} C_VEL
LIN {X 0,Y 728.089,Z 330.527,A -85,B 0,C 180,E1 -1107.657,E2 -1107.657} C_VEL
LIN {X 0,Y 728.1,Z 330.531,A -85,B 0,C 180,E1 -1110.174,E2 -1110.174} C_VEL
LIN {X 0,Y 728.146,Z 330.527,A -85,B 0,C 180,E1 -1113.13,E2 -1113.13} C_VEL
LIN {X 0,Y 728.087,Z 330.53,A -85,B 0,C 180,E1 -1115.805,E2 -1115.805} C_VEL
LIN {X 0,Y 728.106,Z 330.531,A -85,B 0,C 180,E1 -1118.369,E2 -1118.369} C_VEL
LIN {X 0,Y 728.122,Z 330.527,A -85,B 0,C 180,E1 -1121.446,E2 -1121.446} C_VEL
LIN {X 0,Y 728.086,Z 330.53,A -85,B 0,C 180,E1 -1124.09,E2 -1124.09} C_VEL
LIN {X 0,Y 728.131,Z 330.534,A -85,B 0,C 180,E1 -1126.745,E2 -1126.745} C_VEL
LIN {X 0,Y 728.108,Z 330.531,A -85,B 0,C 180,E1 -1129.698,E2 -1129.698} C_VEL
LIN {X 0,Y 728.095,Z 330.601,A -85,B 0,C 180,E1 -1132.253,E2 -1132.253} C_VEL
LIN {X 0,Y 731.737,Z 340.721,A -85,B 0,C 180,E1 -1133.202,E2 -1133.202} C_VEL
LIN {X 0,Y 731.312,Z 376.071,A -85,B 0,C 180,E1 -1135.672,E2 -1135.672} C_VEL
LIN {X 0,Y 731.483,Z 377.843,A -85,B 0,C 180,E1 -1135.757,E2 -1135.757} C_VEL
LIN {X 0,Y 733.119,Z 385.204,A -85,B 0,C 180,E1 -1135.929,E2 -1135.929} C_VEL
LIN {X 0,Y 732.283,Z 644.202,A -85,B 0,C 180,E1 -1138.84,E2 -1138.84} C_VEL
LIN {X 0,Y 731.89,Z 766.852,A -85,B 0,C 180,E1 -1140.213,E2 -1140.213} C_VEL
LIN {X 0,Y 731.63,Z 792.379,A -85,B 0,C 180,E1 -1140.64,E2 -1140.64} C_VEL
LIN {X 0,Y 731.417,Z 813.903,A -85,B 0,C 180,E1 -1141.135,E2 -1141.135} C_VEL
LIN {X 0,Y 731.153,Z 837.29,A -85,B 0,C 180,E1 -1141.804,E2 -1141.804} C_VEL
LIN {X 0,Y 730.784,Z 860.276,A -85,B 0,C 180,E1 -1142.622,E2 -1142.622} C_VEL
LIN {X 0,Y 730.482,Z 882.073,A -85,B 0,C 180,E1 -1143.535,E2 -1143.535} C_VEL
LIN {X 0,Y 730.059,Z 903.946,A -85,B 0,C 180,E1 -1144.616,E2 -1144.616} C_VEL
LIN {X 0,Y 729.749,Z 924.343,A -85,B 0,C 180,E1 -1145.772,E2 -1145.772} C_VEL
LIN {X 0,Y 729.364,Z 944.443,A -85,B 0,C 180,E1 -1147.087,E2 -1147.087} C_VEL
LIN {X 0,Y 729.086,Z 963.251,A -85,B 0,C 180,E1 -1148.478,E2 -1148.478} C_VEL
LIN {X 0,Y 728.782,Z 980.461,A -85,B 0,C 180,E1 -1149.94,E2 -1149.94} C_VEL
LIN {X 0,Y 728.57,Z 996.962,A -85,B 0,C 180,E1 -1151.517,E2 -1151.517} C_VEL
LIN {X 0,Y 728.358,Z 1011.447,A -85,B 0,C 180,E1 -1153.107,E2 -1153.107} C_VEL
LIN {X 0,Y 728.222,Z 1025.058,A -85,B 0,C 180,E1 -1154.796,E2 -1154.796} C_VEL
LIN {X 0,Y 728.102,Z 1036.794,A -85,B 0,C 180,E1 -1156.499,E2 -1156.499} C_VEL
LIN {X 0,Y 728.013,Z 1046.95,A -85,B 0,C 180,E1 -1158.191,E2 -1158.191} C_VEL
LIN {X 0,Y 727.951,Z 1056.181,A -85,B 0,C 180,E1 -1160.034,E2 -1160.034} C_VEL
LIN {X 0,Y 727.929,Z 1062.815,A -85,B 0,C 180,E1 -1161.628,E2 -1161.628} C_VEL
LIN {X 0,Y 727.905,Z 1069.245,A -85,B 0,C 180,E1 -1163.532,E2 -1163.532} C_VEL
LIN {X 0,Y 727.917,Z 1073.654,A -85,B 0,C 180,E1 -1165.351,E2 -1165.351} C_VEL
LIN {X 0,Y 727.911,Z 1076.572,A -85,B 0,C 180,E1 -1167.087,E2 -1167.087} C_VEL
LIN {X 0,Y 727.905,Z 1078.262,A -85,B 0,C 180,E1 -1169.134,E2 -1169.134} C_VEL
LIN {X 0,Y 727.899,Z 1078.284,A -85,B 0,C 180,E1 -1170.787,E2 -1170.787} C_VEL
LIN {X 0,Y 727.906,Z 1076.796,A -85,B 0,C 180,E1 -1172.756,E2 -1172.756} C_VEL
LIN {X 0,Y 727.913,Z 1073.813,A -85,B 0,C 180,E1 -1174.57,E2 -1174.57} C_VEL
LIN {X 0,Y 727.907,Z 1069.451,A -85,B 0,C 180,E1 -1176.388,E2 -1176.388} C_VEL
LIN {X 0,Y 727.935,Z 1063.118,A -85,B 0,C 180,E1 -1178.293,E2 -1178.293} C_VEL
LIN {X 0,Y 727.947,Z 1056.536,A -85,B 0,C 180,E1 -1179.886,E2 -1179.886} C_VEL
LIN {X 0,Y 728.016,Z 1047.41,A -85,B 0,C 180,E1 -1181.728,E2 -1181.728} C_VEL
LIN {X 0,Y 728.099,Z 1037.315,A -85,B 0,C 180,E1 -1183.42,E2 -1183.42} C_VEL
LIN {X 0,Y 728.214,Z 1025.489,A -85,B 0,C 180,E1 -1185.144,E2 -1185.144} C_VEL
LIN {X 0,Y 728.358,Z 1011.926,A -85,B 0,C 180,E1 -1186.838,E2 -1186.838} C_VEL
LIN {X 0,Y 728.547,Z 997.739,A -85,B 0,C 180,E1 -1188.401,E2 -1188.401} C_VEL
LIN {X 0,Y 728.773,Z 981.391,A -85,B 0,C 180,E1 -1189.976,E2 -1189.976} C_VEL
LIN {X 0,Y 729.064,Z 964.272,A -85,B 0,C 180,E1 -1191.438,E2 -1191.438} C_VEL
LIN {X 0,Y 729.347,Z 945.65,A -85,B 0,C 180,E1 -1192.829,E2 -1192.829} C_VEL
LIN {X 0,Y 729.72,Z 926.427,A -85,B 0,C 180,E1 -1194.1,E2 -1194.1} C_VEL
LIN {X 0,Y 730.042,Z 905.214,A -85,B 0,C 180,E1 -1195.316,E2 -1195.316} C_VEL
LIN {X 0,Y 730.442,Z 884.085,A -85,B 0,C 180,E1 -1196.372,E2 -1196.372} C_VEL
LIN {X 0,Y 730.773,Z 861.599,A -85,B 0,C 180,E1 -1197.326,E2 -1197.326} C_VEL
LIN {X 0,Y 731.067,Z 840.358,A -85,B 0,C 180,E1 -1198.093,E2 -1198.093} C_VEL
LIN {X 0,Y 731.41,Z 815.372,A -85,B 0,C 180,E1 -1198.827,E2 -1198.827} C_VEL
LIN {X 0,Y 731.614,Z 794.548,A -85,B 0,C 180,E1 -1199.314,E2 -1199.314} C_VEL
LIN {X 0,Y 731.882,Z 769.639,A -85,B 0,C 180,E1 -1199.751,E2 -1199.751} C_VEL
LIN {X 0,Y 732.058,Z 720.307,A -85,B 0,C 180,E1 -1200.32,E2 -1200.32} C_VEL
LIN {X 0,Y 732.828,Z 469.086,A -85,B 0,C 180,E1 -1203.119,E2 -1203.119} C_VEL
LIN {X 0,Y 732.922,Z 383.497,A -85,B 0,C 180,E1 -1204.101,E2 -1204.101} C_VEL
LIN {X 0,Y 731.303,Z 376.685,A -85,B 0,C 180,E1 -1204.285,E2 -1204.285} C_VEL
LIN {X 0,Y 731.729,Z 341.21,A -85,B 0,C 180,E1 -1206.764,E2 -1206.764} C_VEL
LIN {X 0,Y 730.55,Z 337.116,A -85,B 0,C 180,E1 -1207.127,E2 -1207.127} C_VEL
LIN {X 0,Y 728.085,Z 330.536,A -85,B 0,C 180,E1 -1207.77,E2 -1207.77} C_VEL
LIN {X 0,Y 728.114,Z 330.534,A -85,B 0,C 180,E1 -1210.345,E2 -1210.345} C_VEL
LIN {X 0,Y 728.114,Z 330.534,A -85,B 0,C 180,E1 -1213.41,E2 -1213.41} C_VEL
LIN {X 0,Y 728.085,Z 330.531,A -85,B 0,C 180,E1 -1215.981,E2 -1215.981} C_VEL
LIN {X 0,Y 728.141,Z 330.527,A -85,B 0,C 180,E1 -1218.69,E2 -1218.69} C_VEL
LIN {X 0,Y 728.104,Z 330.531,A -85,B 0,C 180,E1 -1221.641,E2 -1221.641} C_VEL
LIN {X 0,Y 728.087,Z 330.529,A -85,B 0,C 180,E1 -1224.195,E2 -1224.195} C_VEL
LIN {X 0,Y 728.157,Z 330.525,A -85,B 0,C 180,E1 -1226.965,E2 -1226.965} C_VEL
LIN {X 0,Y 728.096,Z 330.53,A -85,B 0,C 180,E1 -1229.903,E2 -1229.903} C_VEL
LIN {X 0,Y 728.091,Z 330.526,A -85,B 0,C 180,E1 -1232.432,E2 -1232.432} C_VEL
LIN {X 0,Y 728.162,Z 330.53,A -85,B 0,C 180,E1 -1235.327,E2 -1235.327} C_VEL
LIN {X 0,Y 728.092,Z 330.531,A -85,B 0,C 180,E1 -1238.066,E2 -1238.066} C_VEL
LIN {X 0,Y 728.091,Z 330.526,A -85,B 0,C 180,E1 -1240.589,E2 -1240.589} C_VEL
LIN {X 0,Y 728.161,Z 330.53,A -85,B 0,C 180,E1 -1243.486,E2 -1243.486} C_VEL
LIN {X 0,Y 728.092,Z 330.529,A -85,B 0,C 180,E1 -1246.256,E2 -1246.256} C_VEL
LIN {X 0,Y 728.094,Z 330.528,A -85,B 0,C 180,E1 -1248.755,E2 -1248.755} C_VEL
LIN {X 0,Y 728.162,Z 330.527,A -85,B 0,C 180,E1 -1251.63,E2 -1251.63} C_VEL
LIN {X 0,Y 728.092,Z 330.528,A -85,B 0,C 180,E1 -1254.404,E2 -1254.404} C_VEL
LIN {X 0,Y 728.098,Z 330.526,A -85,B 0,C 180,E1 -1256.93,E2 -1256.93} C_VEL
LIN {X 0,Y 728.161,Z 330.53,A -85,B 0,C 180,E1 -1259.843,E2 -1259.843} C_VEL
LIN {X 0,Y 728.091,Z 330.53,A -85,B 0,C 180,E1 -1262.598,E2 -1262.598} C_VEL
LIN {X 0,Y 728.108,Z 330.525,A -85,B 0,C 180,E1 -1265.2,E2 -1265.2} C_VEL
LIN {X 0,Y 728.133,Z 330.533,A -85,B 0,C 180,E1 -1268.211,E2 -1268.211} C_VEL
LIN {X 0,Y 728.089,Z 330.525,A -85,B 0,C 180,E1 -1270.914,E2 -1270.914} C_VEL
LIN {X 0,Y 728.13,Z 330.525,A -85,B 0,C 180,E1 -1273.519,E2 -1273.519} C_VEL
LIN {X 0,Y 727.195,Z 330.653,A -85,B 0,C 180,E1 -1274.125,E2 -1274.125} C_VEL
LIN {X 0,Y 720.682,Z 331.459,A -85,B 0,C 180,E1 -1275.866,E2 -1275.866} C_VEL
LIN {X 0,Y 720.206,Z 331.518,A -85,B 0,C 180,E1 -1276.264,E2 -1276.264} C_VEL
LIN {X 0,Y 720.151,Z 331.518,A -85,B 0,C 180,E1 -1278.998,E2 -1278.998} C_VEL
LIN {X 0,Y 720.193,Z 331.511,A -85,B 0,C 180,E1 -1281.673,E2 -1281.673} C_VEL
LIN {X 0,Y 720.17,Z 331.516,A -85,B 0,C 180,E1 -1284.703,E2 -1284.703} C_VEL
LIN {X 0,Y 720.155,Z 331.517,A -85,B 0,C 180,E1 -1287.302,E2 -1287.302} C_VEL
LIN {X 0,Y 720.222,Z 331.512,A -85,B 0,C 180,E1 -1290.127,E2 -1290.127} C_VEL
LIN {X 0,Y 720.159,Z 331.516,A -85,B 0,C 180,E1 -1293.006,E2 -1293.006} C_VEL
LIN {X 0,Y 720.161,Z 331.517,A -85,B 0,C 180,E1 -1295.574,E2 -1295.574} C_VEL
LIN {X 0,Y 720.218,Z 331.522,A -85,B 0,C 180,E1 -1298.562,E2 -1298.562} C_VEL
LIN {X 0,Y 720.154,Z 331.52,A -85,B 0,C 180,E1 -1301.31,E2 -1301.31} C_VEL
LIN {X 0,Y 720.183,Z 331.508,A -85,B 0,C 180,E1 -1303.963,E2 -1303.963} C_VEL
LIN {X 0,Y 720.178,Z 331.52,A -85,B 0,C 180,E1 -1307.028,E2 -1307.028} C_VEL
LIN {X 0,Y 720.156,Z 331.519,A -85,B 0,C 180,E1 -1309.683,E2 -1309.683} C_VEL
LIN {X 0,Y 720.223,Z 331.518,A -85,B 0,C 180,E1 -1312.449,E2 -1312.449} C_VEL
LIN {X 0,Y 720.161,Z 331.526,A -85,B 0,C 180,E1 -1315.398,E2 -1315.398} C_VEL
LIN {X 0,Y 720.177,Z 331.614,A -85,B 0,C 180,E1 -1315.956,E2 -1315.956} C_VEL
LIN {X 0,Y 724.011,Z 342.788,A -85,B 0,C 180,E1 -1317.035,E2 -1317.035} C_VEL
LIN {X 0,Y 724.098,Z 347.958,A -85,B 0,C 180,E1 -1317.405,E2 -1317.405} C_VEL
LIN {X 0,Y 726.437,Z 357.404,A -85,B 0,C 180,E1 -1317.643,E2 -1317.643} C_VEL
LIN {X 0,Y 725.512,Z 593.015,A -85,B 0,C 180,E1 -1320.32,E2 -1320.32} C_VEL
LIN {X 0,Y 724.937,Z 736.823,A -85,B 0,C 180,E1 -1321.943,E2 -1321.943} C_VEL
LIN {X 0,Y 724.624,Z 762.352,A -85,B 0,C 180,E1 -1322.373,E2 -1322.373} C_VEL
LIN {X 0,Y 724.346,Z 784.069,A -85,B 0,C 180,E1 -1322.876,E2 -1322.876} C_VEL
LIN {X 0,Y 724.009,Z 807.47,A -85,B 0,C 180,E1 -1323.552,E2 -1323.552} C_VEL
LIN {X 0,Y 723.551,Z 830.3,A -85,B 0,C 180,E1 -1324.371,E2 -1324.371} C_VEL
LIN {X 0,Y 723.158,Z 852.703,A -85,B 0,C 180,E1 -1325.319,E2 -1325.319} C_VEL
LIN {X 0,Y 722.63,Z 874.823,A -85,B 0,C 180,E1 -1326.429,E2 -1326.429} C_VEL
LIN {X 0,Y 722.214,Z 895.894,A -85,B 0,C 180,E1 -1327.644,E2 -1327.644} C_VEL
LIN {X 0,Y 721.757,Z 915.307,A -85,B 0,C 180,E1 -1328.938,E2 -1328.938} C_VEL
LIN {X 0,Y 721.375,Z 934.393,A -85,B 0,C 180,E1 -1330.377,E2 -1330.377} C_VEL
LIN {X 0,Y 721.013,Z 951.109,A -85,B 0,C 180,E1 -1331.819,E2 -1331.819} C_VEL
LIN {X 0,Y 720.724,Z 968.107,A -85,B 0,C 180,E1 -1333.477,E2 -1333.477} C_VEL
LIN {X 0,Y 720.471,Z 982.124,A -85,B 0,C 180,E1 -1335.041,E2 -1335.041} C_VEL
LIN {X 0,Y 720.277,Z 996.262,A -85,B 0,C 180,E1 -1336.84,E2 -1336.84} C_VEL
LIN {X 0,Y 720.145,Z 1007.27,A -85,B 0,C 180,E1 -1338.467,E2 -1338.467} C_VEL
LIN {X 0,Y 720.051,Z 1018.192,A -85,B 0,C 180,E1 -1340.327,E2 -1340.327} C_VEL
LIN {X 0,Y 719.965,Z 1026.754,A -85,B 0,C 180,E1 -1342.097,E2 -1342.097} C_VEL
LIN {X 0,Y 719.945,Z 1033.577,A -85,B 0,C 180,E1 -1343.781,E2 -1343.781} C_VEL
LIN {X 0,Y 719.92,Z 1039.949,A -85,B 0,C 180,E1 -1345.779,E2 -1345.779} C_VEL
LIN {X 0,Y 719.916,Z 1044.027,A -85,B 0,C 180,E1 -1347.532,E2 -1347.532} C_VEL
LIN {X 0,Y 719.896,Z 1047.044,A -85,B 0,C 180,E1 -1349.443,E2 -1349.443} C_VEL
LIN {X 0,Y 719.893,Z 1048.313,A -85,B 0,C 180,E1 -1351.353,E2 -1351.353} C_VEL
LIN {X 0,Y 719.911,Z 1048.21,A -85,B 0,C 180,E1 -1353.105,E2 -1353.105} C_VEL
LIN {X 0,Y 719.913,Z 1046.418,A -85,B 0,C 180,E1 -1355.1,E2 -1355.1} C_VEL
LIN {X 0,Y 719.909,Z 1043.586,A -85,B 0,C 180,E1 -1356.78,E2 -1356.78} C_VEL
LIN {X 0,Y 719.918,Z 1038.879,A -85,B 0,C 180,E1 -1358.707,E2 -1358.707} C_VEL
LIN {X 0,Y 719.933,Z 1032.921,A -85,B 0,C 180,E1 -1360.483,E2 -1360.483} C_VEL
LIN {X 0,Y 719.978,Z 1026.19,A -85,B 0,C 180,E1 -1362.121,E2 -1362.121} C_VEL
LIN {X 0,Y 720.061,Z 1016.044,A -85,B 0,C 180,E1 -1364.146,E2 -1364.146} C_VEL
LIN {X 0,Y 720.162,Z 1006.099,A -85,B 0,C 180,E1 -1365.807,E2 -1365.807} C_VEL
LIN {X 0,Y 720.325,Z 993.579,A -85,B 0,C 180,E1 -1367.614,E2 -1367.614} C_VEL
LIN {X 0,Y 720.485,Z 980.819,A -85,B 0,C 180,E1 -1369.203,E2 -1369.203} C_VEL
LIN {X 0,Y 720.775,Z 965.502,A -85,B 0,C 180,E1 -1370.887,E2 -1370.887} C_VEL
LIN {X 0,Y 721.067,Z 949.122,A -85,B 0,C 180,E1 -1372.451,E2 -1372.451} C_VEL
LIN {X 0,Y 721.435,Z 931.29,A -85,B 0,C 180,E1 -1373.959,E2 -1373.959} C_VEL
LIN {X 0,Y 721.816,Z 913.167,A -85,B 0,C 180,E1 -1375.303,E2 -1375.303} C_VEL
LIN {X 0,Y 722.27,Z 891.782,A -85,B 0,C 180,E1 -1376.694,E2 -1376.694} C_VEL
LIN {X 0,Y 722.701,Z 872.392,A -85,B 0,C 180,E1 -1377.791,E2 -1377.791} C_VEL
LIN {X 0,Y 723.201,Z 848.869,A -85,B 0,C 180,E1 -1378.941,E2 -1378.941} C_VEL
LIN {X 0,Y 723.594,Z 828.32,A -85,B 0,C 180,E1 -1379.796,E2 -1379.796} C_VEL
LIN {X 0,Y 724.064,Z 803.979,A -85,B 0,C 180,E1 -1380.646,E2 -1380.646} C_VEL
LIN {X 0,Y 724.363,Z 781.807,A -85,B 0,C 180,E1 -1381.273,E2 -1381.273} C_VEL
LIN {X 0,Y 724.745,Z 757.551,A -85,B 0,C 180,E1 -1381.813,E2 -1381.813} C_VEL
LIN {X 0,Y 724.949,Z 734.194,A -85,B 0,C 180,E1 -1382.182,E2 -1382.182} C_VEL
LIN {X 0,Y 725.996,Z 471.715,A -85,B 0,C 180,E1 -1385.139,E2 -1385.139} C_VEL
LIN {X 0,Y 726.255,Z 355.961,A -85,B 0,C 180,E1 -1386.474,E2 -1386.474} C_VEL
LIN {X 0,Y 723.986,Z 347.403,A -85,B 0,C 180,E1 -1386.705,E2 -1386.705} C_VEL
LIN {X 0,Y 723.878,Z 342.446,A -85,B 0,C 180,E1 -1387.089,E2 -1387.089} C_VEL
LIN {X 0,Y 720.162,Z 331.525,A -85,B 0,C 180,E1 -1388.159,E2 -1388.159} C_VEL
LIN {X 0,Y 720.159,Z 331.524,A -85,B 0,C 180,E1 -1390.735,E2 -1390.735} C_VEL
LIN {X 0,Y 720.222,Z 331.515,A -85,B 0,C 180,E1 -1393.671,E2 -1393.671} C_VEL
LIN {X 0,Y 720.153,Z 331.517,A -85,B 0,C 180,E1 -1396.475,E2 -1396.475} C_VEL
LIN {X 0,Y 720.171,Z 331.518,A -85,B 0,C 180,E1 -1399.055,E2 -1399.055} C_VEL
LIN {X 0,Y 720.182,Z 331.515,A -85,B 0,C 180,E1 -1402.145,E2 -1402.145} C_VEL
LIN {X 0,Y 720.151,Z 331.51,A -85,B 0,C 180,E1 -1404.816,E2 -1404.816} C_VEL
LIN {X 0,Y 720.219,Z 331.52,A -85,B 0,C 180,E1 -1407.596,E2 -1407.596} C_VEL
LIN {X 0,Y 720.16,Z 331.517,A -85,B 0,C 180,E1 -1410.522,E2 -1410.522} C_VEL
LIN {X 0,Y 720.158,Z 331.519,A -85,B 0,C 180,E1 -1413.087,E2 -1413.087} C_VEL
LIN {X 0,Y 720.223,Z 331.516,A -85,B 0,C 180,E1 -1415.998,E2 -1415.998} C_VEL
LIN {X 0,Y 720.153,Z 331.515,A -85,B 0,C 180,E1 -1418.839,E2 -1418.839} C_VEL
LIN {X 0,Y 720.174,Z 331.521,A -85,B 0,C 180,E1 -1421.461,E2 -1421.461} C_VEL
LIN {X 0,Y 720.178,Z 331.515,A -85,B 0,C 180,E1 -1424.54,E2 -1424.54} C_VEL
LIN {X 0,Y 720.151,Z 331.517,A -85,B 0,C 180,E1 -1427.164,E2 -1427.164} C_VEL
LIN {X 0,Y 720.215,Z 331.519,A -85,B 0,C 180,E1 -1429.925,E2 -1429.925} C_VEL
LIN {X 0,Y 720.158,Z 331.516,A -85,B 0,C 180,E1 -1432.902,E2 -1432.902} C_VEL
LIN {X 0,Y 720.157,Z 331.518,A -85,B 0,C 180,E1 -1435.484,E2 -1435.484} C_VEL
LIN {X 0,Y 720.221,Z 331.513,A -85,B 0,C 180,E1 -1438.409,E2 -1438.409} C_VEL
LIN {X 0,Y 720.151,Z 331.518,A -85,B 0,C 180,E1 -1441.193,E2 -1441.193} C_VEL
LIN {X 0,Y 720.171,Z 331.518,A -85,B 0,C 180,E1 -1443.821,E2 -1443.821} C_VEL
LIN {X 0,Y 720.174,Z 331.512,A -85,B 0,C 180,E1 -1446.938,E2 -1446.938} C_VEL
LIN {X 0,Y 720.149,Z 331.519,A -85,B 0,C 180,E1 -1449.51,E2 -1449.51} C_VEL
LIN {X 0,Y 720.21,Z 331.518,A -85,B 0,C 180,E1 -1452.264,E2 -1452.264} C_VEL
LIN {X 0,Y 720.162,Z 331.513,A -85,B 0,C 180,E1 -1455.214,E2 -1455.214} C_VEL
LIN {X 0,Y 720.152,Z 331.519,A -85,B 0,C 180,E1 -1457.786,E2 -1457.786} C_VEL
LIN {X 0,Y 720.223,Z 331.518,A -85,B 0,C 180,E1 -1460.656,E2 -1460.656} C_VEL
LIN {X 0,Y 720.153,Z 331.514,A -85,B 0,C 180,E1 -1463.483,E2 -1463.483} C_VEL
LIN {X 0,Y 720.156,Z 331.52,A -85,B 0,C 180,E1 -1466.024,E2 -1466.024} C_VEL
LIN {X 0,Y 720.219,Z 331.514,A -85,B 0,C 180,E1 -1468.998,E2 -1468.998} C_VEL
